			//Surplus
			IF bSurplusAvailable AND Lynus_Standards.GVL_Energy.stDataElectricHeatingElements[diNrOfEMS_OUT,arrCTCheckActivePrio[3]].byPriority = arrActualPrioInTurn[3] AND NOT Lynus_Standards.GVL_Energy.stDataElectricHeatingElements[diNrOfEMS_OUT,arrCTCheckActivePrio[3]].bIsStepSwitched AND NOT 
				Lynus_Standards.GVL_Energy.stDataElectricHeatingElements[diNrOfEMS_OUT,arrCTCheckActivePrio[3]].bIsControllable AND Lynus_Standards.GVL_Energy.stDataElectricHeatingElements[diNrOfEMS_OUT,arrCTCheckActivePrio[3]].arrTargetPowerEMS[1] < 100 THEN
					arrActualStepInTurn[2] := 1;	
						arrMaxPrioReached[3] := FALSE;
							arrMinPrioReached[3] := FALSE;
								arrCTCheckActivePrio[3] := 0;
									uiState := 90;
			ELSIF bSurplusAvailable AND Lynus_Standards.GVL_Energy.stDataElectricHeatingElements[diNrOfEMS_OUT,arrCTCheckActivePrio[3]].byPriority = arrActualPrioInTurn[3] AND Lynus_Standards.GVL_Energy.stDataElectricHeatingElements[diNrOfEMS_OUT,arrCTCheckActivePrio[3]].byNumberOfSteps = 0 AND
				Lynus_Standards.GVL_Energy.stDataElectricHeatingElements[diNrOfEMS_OUT,arrCTCheckActivePrio[3]].arrTargetPowerEMS[1] < 100 THEN 
					arrActualStepInTurn[2] := 1;	
						arrMaxPrioReached[3] := FALSE;
							arrMinPrioReached[3] := FALSE;
								arrCTCheckActivePrio[3] := 0;
									uiState := 90;
			ELSIF bSurplusAvailable AND Lynus_Standards.GVL_Energy.stDataElectricHeatingElements[diNrOfEMS_OUT,arrCTCheckActivePrio[3]].byPriority = arrActualPrioInTurn[3] AND NOT Lynus_Standards.GVL_Energy.stDataElectricHeatingElements[diNrOfEMS_OUT,arrCTCheckActivePrio[3]].bIsStepSwitched AND 
				Lynus_Standards.GVL_Energy.stDataElectricHeatingElements[diNrOfEMS_OUT,arrCTCheckActivePrio[3]].bIsControllable AND Lynus_Standards.GVL_Energy.stDataElectricHeatingElements[diNrOfEMS_OUT,arrCTCheckActivePrio[3]].arrTargetPowerEMS[1] < 100 THEN
					arrActualStepInTurn[2] := 1;	
						arrMaxPrioReached[3] := FALSE;
							arrMinPrioReached[3] := FALSE;
								arrCTCheckActivePrio[3] := 0;
									uiState := 90;	
			ELSIF bSurplusAvailable AND Lynus_Standards.GVL_Energy.stDataElectricHeatingElements[diNrOfEMS_OUT,arrCTCheckActivePrio[3]].byPriority = arrActualPrioInTurn[3] AND Lynus_Standards.GVL_Energy.stDataElectricHeatingElements[diNrOfEMS_OUT,arrCTCheckActivePrio[3]].bIsStepSwitched AND 
				Lynus_Standards.GVL_Energy.stDataElectricHeatingElements[diNrOfEMS_OUT,arrCTCheckActivePrio[3]].bIsControllable AND Lynus_Standards.GVL_Energy.stDataElectricHeatingElements[diNrOfEMS_OUT,arrCTCheckActivePrio[3]].byNumberOfSteps = 1 AND Lynus_Standards.GVL_Energy.stDataElectricHeatingElements[diNrOfEMS_OUT,arrCTCheckActivePrio[3]].arrTargetPowerEMS[1] < 100 THEN 
					arrActualStepInTurn[2] := 1;	
						arrMaxPrioReached[3] := FALSE;
							arrMinPrioReached[3] := FALSE;
								arrCTCheckActivePrio[3] := 0;
									uiState := 90;
			ELSIF bSurplusAvailable AND Lynus_Standards.GVL_Energy.stDataElectricHeatingElements[diNrOfEMS_OUT,arrCTCheckActivePrio[3]].byPriority = arrActualPrioInTurn[3] AND Lynus_Standards.GVL_Energy.stDataElectricHeatingElements[diNrOfEMS_OUT,arrCTCheckActivePrio[3]].bIsStepSwitched AND 
				Lynus_Standards.GVL_Energy.stDataElectricHeatingElements[diNrOfEMS_OUT,arrCTCheckActivePrio[3]].bIsControllable AND Lynus_Standards.GVL_Energy.stDataElectricHeatingElements[diNrOfEMS_OUT,arrCTCheckActivePrio[3]].byNumberOfSteps = 2 AND (Lynus_Standards.GVL_Energy.stDataElectricHeatingElements[diNrOfEMS_OUT,arrCTCheckActivePrio[3]].arrTargetPowerEMS[1] < 100 OR Lynus_Standards.GVL_Energy.stDataElectricHeatingElements[diNrOfEMS_OUT,arrCTCheckActivePrio[3]].arrTargetPowerEMS[2] < 100) THEN
					IF Lynus_Standards.GVL_Energy.stDataElectricHeatingElements[diNrOfEMS_OUT,arrCTCheckActivePrio[3]].arrTargetPowerEMS[1] >= 100 THEN arrActualStepInTurn[2] := 2; ELSE arrActualStepInTurn[2] := 1; END_IF
						arrMaxPrioReached[3] := FALSE;
							arrMinPrioReached[3] := FALSE;
								arrCTCheckActivePrio[3] := 0;
									uiState := 90;
			ELSIF bSurplusAvailable AND Lynus_Standards.GVL_Energy.stDataElectricHeatingElements[diNrOfEMS_OUT,arrCTCheckActivePrio[3]].byPriority = arrActualPrioInTurn[3] AND Lynus_Standards.GVL_Energy.stDataElectricHeatingElements[diNrOfEMS_OUT,arrCTCheckActivePrio[3]].bIsStepSwitched AND 
				Lynus_Standards.GVL_Energy.stDataElectricHeatingElements[diNrOfEMS_OUT,arrCTCheckActivePrio[3]].bIsControllable AND Lynus_Standards.GVL_Energy.stDataElectricHeatingElements[diNrOfEMS_OUT,arrCTCheckActivePrio[3]].byNumberOfSteps = 3 AND (Lynus_Standards.GVL_Energy.stDataElectricHeatingElements[diNrOfEMS_OUT,arrCTCheckActivePrio[3]].arrTargetPowerEMS[1] < 100 OR Lynus_Standards.GVL_Energy.stDataElectricHeatingElements[diNrOfEMS_OUT,arrCTCheckActivePrio[3]].arrTargetPowerEMS[2] < 100 OR Lynus_Standards.GVL_Energy.stDataElectricHeatingElements[diNrOfEMS_OUT,arrCTCheckActivePrio[3]].arrTargetPowerEMS[3] < 100) THEN
					IF Lynus_Standards.GVL_Energy.stDataElectricHeatingElements[diNrOfEMS_OUT,arrCTCheckActivePrio[3]].arrTargetPowerEMS[1] < 100 THEN arrActualStepInTurn[2] := 1; END_IF
					IF Lynus_Standards.GVL_Energy.stDataElectricHeatingElements[diNrOfEMS_OUT,arrCTCheckActivePrio[3]].arrTargetPowerEMS[1] >= 100 THEN arrActualStepInTurn[2] := 2; END_IF
					IF Lynus_Standards.GVL_Energy.stDataElectricHeatingElements[diNrOfEMS_OUT,arrCTCheckActivePrio[3]].arrTargetPowerEMS[2] >= 100 THEN arrActualStepInTurn[2] := 3; END_IF
						arrMaxPrioReached[3] := FALSE;
							arrMinPrioReached[3] := FALSE;
								arrCTCheckActivePrio[3] := 0;
									uiState := 90;
			ELSIF bSurplusAvailable AND Lynus_Standards.GVL_Energy.stDataElectricHeatingElements[diNrOfEMS_OUT,arrCTCheckActivePrio[3]].byPriority = arrActualPrioInTurn[3] AND Lynus_Standards.GVL_Energy.stDataElectricHeatingElements[diNrOfEMS_OUT,arrCTCheckActivePrio[3]].bIsStepSwitched AND 
				Lynus_Standards.GVL_Energy.stDataElectricHeatingElements[diNrOfEMS_OUT,arrCTCheckActivePrio[3]].bIsControllable AND Lynus_Standards.GVL_Energy.stDataElectricHeatingElements[diNrOfEMS_OUT,arrCTCheckActivePrio[3]].byNumberOfSteps = 4 AND 
					(Lynus_Standards.GVL_Energy.stDataElectricHeatingElements[diNrOfEMS_OUT,arrCTCheckActivePrio[3]].arrTargetPowerEMS[1] < 100 OR Lynus_Standards.GVL_Energy.stDataElectricHeatingElements[diNrOfEMS_OUT,arrCTCheckActivePrio[3]].arrTargetPowerEMS[2] < 100 OR Lynus_Standards.GVL_Energy.stDataElectricHeatingElements[diNrOfEMS_OUT,arrCTCheckActivePrio[3]].arrTargetPowerEMS[3] < 100 OR
						Lynus_Standards.GVL_Energy.stDataElectricHeatingElements[diNrOfEMS_OUT,arrCTCheckActivePrio[3]].arrTargetPowerEMS[4] < 100) THEN
							IF Lynus_Standards.GVL_Energy.stDataElectricHeatingElements[diNrOfEMS_OUT,arrCTCheckActivePrio[3]].arrTargetPowerEMS[1] < 100 THEN arrActualStepInTurn[2] := 1; END_IF
							IF Lynus_Standards.GVL_Energy.stDataElectricHeatingElements[diNrOfEMS_OUT,arrCTCheckActivePrio[3]].arrTargetPowerEMS[1] >= 100 THEN arrActualStepInTurn[2] := 2; END_IF
							IF Lynus_Standards.GVL_Energy.stDataElectricHeatingElements[diNrOfEMS_OUT,arrCTCheckActivePrio[3]].arrTargetPowerEMS[2] >= 100 THEN arrActualStepInTurn[2] := 3; END_IF
							IF Lynus_Standards.GVL_Energy.stDataElectricHeatingElements[diNrOfEMS_OUT,arrCTCheckActivePrio[3]].arrTargetPowerEMS[3] >= 100 THEN arrActualStepInTurn[2] := 4; END_IF
								arrMaxPrioReached[3] := FALSE;
									arrMinPrioReached[3] := FALSE;
										arrCTCheckActivePrio[3] := 0;
											uiState := 90;
			ELSIF bSurplusAvailable AND Lynus_Standards.GVL_Energy.stDataElectricHeatingElements[diNrOfEMS_OUT,arrCTCheckActivePrio[3]].byPriority = arrActualPrioInTurn[3] AND Lynus_Standards.GVL_Energy.stDataElectricHeatingElements[diNrOfEMS_OUT,arrCTCheckActivePrio[3]].bIsStepSwitched AND 
				Lynus_Standards.GVL_Energy.stDataElectricHeatingElements[diNrOfEMS_OUT,arrCTCheckActivePrio[3]].bIsControllable AND Lynus_Standards.GVL_Energy.stDataElectricHeatingElements[diNrOfEMS_OUT,arrCTCheckActivePrio[3]].byNumberOfSteps = 5 AND 
					(Lynus_Standards.GVL_Energy.stDataElectricHeatingElements[diNrOfEMS_OUT,arrCTCheckActivePrio[3]].arrTargetPowerEMS[1] < 100 OR Lynus_Standards.GVL_Energy.stDataElectricHeatingElements[diNrOfEMS_OUT,arrCTCheckActivePrio[3]].arrTargetPowerEMS[2] < 100 OR Lynus_Standards.GVL_Energy.stDataElectricHeatingElements[diNrOfEMS_OUT,arrCTCheckActivePrio[3]].arrTargetPowerEMS[3] < 100 OR
						Lynus_Standards.GVL_Energy.stDataElectricHeatingElements[diNrOfEMS_OUT,arrCTCheckActivePrio[3]].arrTargetPowerEMS[4] < 100 OR Lynus_Standards.GVL_Energy.stDataElectricHeatingElements[diNrOfEMS_OUT,arrCTCheckActivePrio[3]].arrTargetPowerEMS[5] < 100) THEN
							IF Lynus_Standards.GVL_Energy.stDataElectricHeatingElements[diNrOfEMS_OUT,arrCTCheckActivePrio[3]].arrTargetPowerEMS[1] < 100 THEN arrActualStepInTurn[2] := 1; END_IF
							IF Lynus_Standards.GVL_Energy.stDataElectricHeatingElements[diNrOfEMS_OUT,arrCTCheckActivePrio[3]].arrTargetPowerEMS[1] >= 100 THEN arrActualStepInTurn[2] := 2; END_IF
							IF Lynus_Standards.GVL_Energy.stDataElectricHeatingElements[diNrOfEMS_OUT,arrCTCheckActivePrio[3]].arrTargetPowerEMS[2] >= 100 THEN arrActualStepInTurn[2] := 3; END_IF
							IF Lynus_Standards.GVL_Energy.stDataElectricHeatingElements[diNrOfEMS_OUT,arrCTCheckActivePrio[3]].arrTargetPowerEMS[3] >= 100 THEN arrActualStepInTurn[2] := 4; END_IF
							IF Lynus_Standards.GVL_Energy.stDataElectricHeatingElements[diNrOfEMS_OUT,arrCTCheckActivePrio[3]].arrTargetPowerEMS[4] >= 100 THEN arrActualStepInTurn[2] := 5; END_IF
								arrMaxPrioReached[3] := FALSE;
									arrMinPrioReached[3] := FALSE;
										arrCTCheckActivePrio[3] := 0;
											uiState := 90;
			ELSIF bSurplusAvailable AND Lynus_Standards.GVL_Energy.stDataElectricHeatingElements[diNrOfEMS_OUT,arrCTCheckActivePrio[3]].byPriority = arrActualPrioInTurn[3] AND Lynus_Standards.GVL_Energy.stDataElectricHeatingElements[diNrOfEMS_OUT,arrCTCheckActivePrio[3]].bIsStepSwitched AND 
				Lynus_Standards.GVL_Energy.stDataElectricHeatingElements[diNrOfEMS_OUT,arrCTCheckActivePrio[3]].bIsControllable AND Lynus_Standards.GVL_Energy.stDataElectricHeatingElements[diNrOfEMS_OUT,arrCTCheckActivePrio[3]].byNumberOfSteps = 6 AND 
					(Lynus_Standards.GVL_Energy.stDataElectricHeatingElements[diNrOfEMS_OUT,arrCTCheckActivePrio[3]].arrTargetPowerEMS[1] < 100 OR Lynus_Standards.GVL_Energy.stDataElectricHeatingElements[diNrOfEMS_OUT,arrCTCheckActivePrio[3]].arrTargetPowerEMS[2]< 100 OR Lynus_Standards.GVL_Energy.stDataElectricHeatingElements[diNrOfEMS_OUT,arrCTCheckActivePrio[3]].arrTargetPowerEMS[3]< 100 OR
						Lynus_Standards.GVL_Energy.stDataElectricHeatingElements[diNrOfEMS_OUT,arrCTCheckActivePrio[3]].arrTargetPowerEMS[4] < 100 OR Lynus_Standards.GVL_Energy.stDataElectricHeatingElements[diNrOfEMS_OUT,arrCTCheckActivePrio[3]].arrTargetPowerEMS[5] < 100 OR Lynus_Standards.GVL_Energy.stDataElectricHeatingElements[diNrOfEMS_OUT,arrCTCheckActivePrio[3]].arrTargetPowerEMS[6] < 100) THEN
							IF Lynus_Standards.GVL_Energy.stDataElectricHeatingElements[diNrOfEMS_OUT,arrCTCheckActivePrio[3]].arrTargetPowerEMS[1] < 100 THEN arrActualStepInTurn[2] := 1; END_IF
							IF Lynus_Standards.GVL_Energy.stDataElectricHeatingElements[diNrOfEMS_OUT,arrCTCheckActivePrio[3]].arrTargetPowerEMS[1] >= 100 THEN arrActualStepInTurn[2] := 2; END_IF
							IF Lynus_Standards.GVL_Energy.stDataElectricHeatingElements[diNrOfEMS_OUT,arrCTCheckActivePrio[3]].arrTargetPowerEMS[2] >= 100 THEN arrActualStepInTurn[2] := 3; END_IF
							IF Lynus_Standards.GVL_Energy.stDataElectricHeatingElements[diNrOfEMS_OUT,arrCTCheckActivePrio[3]].arrTargetPowerEMS[3] >= 100 THEN arrActualStepInTurn[2] := 4; END_IF
							IF Lynus_Standards.GVL_Energy.stDataElectricHeatingElements[diNrOfEMS_OUT,arrCTCheckActivePrio[3]].arrTargetPowerEMS[4] >= 100 THEN arrActualStepInTurn[2] := 5; END_IF
							IF Lynus_Standards.GVL_Energy.stDataElectricHeatingElements[diNrOfEMS_OUT,arrCTCheckActivePrio[3]].arrTargetPowerEMS[5] >= 100 THEN arrActualStepInTurn[2] := 6; END_IF
								arrMaxPrioReached[3] := FALSE;
									arrMinPrioReached[3] := FALSE;
										arrCTCheckActivePrio[3] := 0;
											uiState := 90;
			ELSIF bSurplusAvailable AND Lynus_Standards.GVL_Energy.stDataElectricHeatingElements[diNrOfEMS_OUT,arrCTCheckActivePrio[3]].byPriority = arrActualPrioInTurn[3] AND Lynus_Standards.GVL_Energy.stDataElectricHeatingElements[diNrOfEMS_OUT,arrCTCheckActivePrio[3]].bIsStepSwitched AND 
				Lynus_Standards.GVL_Energy.stDataElectricHeatingElements[diNrOfEMS_OUT,arrCTCheckActivePrio[3]].bIsControllable AND Lynus_Standards.GVL_Energy.stDataElectricHeatingElements[diNrOfEMS_OUT,arrCTCheckActivePrio[3]].byNumberOfSteps= 7 AND 
					(Lynus_Standards.GVL_Energy.stDataElectricHeatingElements[diNrOfEMS_OUT,arrCTCheckActivePrio[3]].arrTargetPowerEMS[1] < 100 OR Lynus_Standards.GVL_Energy.stDataElectricHeatingElements[diNrOfEMS_OUT,arrCTCheckActivePrio[3]].arrTargetPowerEMS[2] < 100 OR Lynus_Standards.GVL_Energy.stDataElectricHeatingElements[diNrOfEMS_OUT,arrCTCheckActivePrio[3]].arrTargetPowerEMS[3] < 100 OR
						Lynus_Standards.GVL_Energy.stDataElectricHeatingElements[diNrOfEMS_OUT,arrCTCheckActivePrio[3]].arrTargetPowerEMS[4] < 100 OR Lynus_Standards.GVL_Energy.stDataElectricHeatingElements[diNrOfEMS_OUT,arrCTCheckActivePrio[3]].arrTargetPowerEMS[5] < 100 OR Lynus_Standards.GVL_Energy.stDataElectricHeatingElements[diNrOfEMS_OUT,arrCTCheckActivePrio[3]].arrTargetPowerEMS[6] < 100 OR
							Lynus_Standards.GVL_Energy.stDataElectricHeatingElements[diNrOfEMS_OUT,arrCTCheckActivePrio[3]].arrTargetPowerEMS[7] < 100) THEN
								IF Lynus_Standards.GVL_Energy.stDataElectricHeatingElements[diNrOfEMS_OUT,arrCTCheckActivePrio[3]].arrTargetPowerEMS[1] < 100 THEN arrActualStepInTurn[2] := 1; END_IF
								IF Lynus_Standards.GVL_Energy.stDataElectricHeatingElements[diNrOfEMS_OUT,arrCTCheckActivePrio[3]].arrTargetPowerEMS[1] >= 100 THEN arrActualStepInTurn[2] := 2; END_IF
								IF Lynus_Standards.GVL_Energy.stDataElectricHeatingElements[diNrOfEMS_OUT,arrCTCheckActivePrio[3]].arrTargetPowerEMS[2] >= 100 THEN arrActualStepInTurn[2] := 3; END_IF
								IF Lynus_Standards.GVL_Energy.stDataElectricHeatingElements[diNrOfEMS_OUT,arrCTCheckActivePrio[3]].arrTargetPowerEMS[3] >= 100 THEN arrActualStepInTurn[2] := 4; END_IF
								IF Lynus_Standards.GVL_Energy.stDataElectricHeatingElements[diNrOfEMS_OUT,arrCTCheckActivePrio[3]].arrTargetPowerEMS[4] >= 100 THEN arrActualStepInTurn[2] := 5; END_IF
								IF Lynus_Standards.GVL_Energy.stDataElectricHeatingElements[diNrOfEMS_OUT,arrCTCheckActivePrio[3]].arrTargetPowerEMS[5] >= 100 THEN arrActualStepInTurn[2] := 6; END_IF
								IF Lynus_Standards.GVL_Energy.stDataElectricHeatingElements[diNrOfEMS_OUT,arrCTCheckActivePrio[3]].arrTargetPowerEMS[6] >= 100 THEN arrActualStepInTurn[2] := 7; END_IF
									arrMaxPrioReached[3] := FALSE;
										arrMinPrioReached[3] := FALSE;
											arrCTCheckActivePrio[3] := 0;
												uiState := 90;
			ELSIF bSurplusAvailable AND Lynus_Standards.GVL_Energy.stDataElectricHeatingElements[diNrOfEMS_OUT,arrCTCheckActivePrio[3]].byPriority = arrActualPrioInTurn[3] AND Lynus_Standards.GVL_Energy.stDataElectricHeatingElements[diNrOfEMS_OUT,arrCTCheckActivePrio[3]].bIsStepSwitched AND 
				Lynus_Standards.GVL_Energy.stDataElectricHeatingElements[diNrOfEMS_OUT,arrCTCheckActivePrio[3]].bIsControllable AND Lynus_Standards.GVL_Energy.stDataElectricHeatingElements[diNrOfEMS_OUT,arrCTCheckActivePrio[3]].byNumberOfSteps = 8 AND 
					(Lynus_Standards.GVL_Energy.stDataElectricHeatingElements[diNrOfEMS_OUT,arrCTCheckActivePrio[3]].arrTargetPowerEMS[1] < 100 OR Lynus_Standards.GVL_Energy.stDataElectricHeatingElements[diNrOfEMS_OUT,arrCTCheckActivePrio[3]].arrTargetPowerEMS[2] < 100 OR Lynus_Standards.GVL_Energy.stDataElectricHeatingElements[diNrOfEMS_OUT,arrCTCheckActivePrio[3]].arrTargetPowerEMS[3] < 100 OR
						Lynus_Standards.GVL_Energy.stDataElectricHeatingElements[diNrOfEMS_OUT,arrCTCheckActivePrio[3]].arrTargetPowerEMS[4] < 100 OR Lynus_Standards.GVL_Energy.stDataElectricHeatingElements[diNrOfEMS_OUT,arrCTCheckActivePrio[3]].arrTargetPowerEMS[5] < 100 OR Lynus_Standards.GVL_Energy.stDataElectricHeatingElements[diNrOfEMS_OUT,arrCTCheckActivePrio[3]].arrTargetPowerEMS[6] < 100 OR
							Lynus_Standards.GVL_Energy.stDataElectricHeatingElements[diNrOfEMS_OUT,arrCTCheckActivePrio[3]].arrTargetPowerEMS[7] < 100 OR Lynus_Standards.GVL_Energy.stDataElectricHeatingElements[diNrOfEMS_OUT,arrCTCheckActivePrio[3]].arrTargetPowerEMS[8] < 100) THEN
								IF Lynus_Standards.GVL_Energy.stDataElectricHeatingElements[diNrOfEMS_OUT,arrCTCheckActivePrio[3]].arrTargetPowerEMS[1] < 100 THEN arrActualStepInTurn[2] := 1; END_IF
								IF Lynus_Standards.GVL_Energy.stDataElectricHeatingElements[diNrOfEMS_OUT,arrCTCheckActivePrio[3]].arrTargetPowerEMS[1] >= 100 THEN arrActualStepInTurn[2] := 2; END_IF
								IF Lynus_Standards.GVL_Energy.stDataElectricHeatingElements[diNrOfEMS_OUT,arrCTCheckActivePrio[3]].arrTargetPowerEMS[2] >= 100 THEN arrActualStepInTurn[2] := 3; END_IF
								IF Lynus_Standards.GVL_Energy.stDataElectricHeatingElements[diNrOfEMS_OUT,arrCTCheckActivePrio[3]].arrTargetPowerEMS[3] >= 100 THEN arrActualStepInTurn[2] := 4; END_IF
								IF Lynus_Standards.GVL_Energy.stDataElectricHeatingElements[diNrOfEMS_OUT,arrCTCheckActivePrio[3]].arrTargetPowerEMS[4] >= 100 THEN arrActualStepInTurn[2] := 5; END_IF
								IF Lynus_Standards.GVL_Energy.stDataElectricHeatingElements[diNrOfEMS_OUT,arrCTCheckActivePrio[3]].arrTargetPowerEMS[5] >= 100 THEN arrActualStepInTurn[2] := 6; END_IF
								IF Lynus_Standards.GVL_Energy.stDataElectricHeatingElements[diNrOfEMS_OUT,arrCTCheckActivePrio[3]].arrTargetPowerEMS[6] >= 100 THEN arrActualStepInTurn[2] := 7; END_IF
								IF Lynus_Standards.GVL_Energy.stDataElectricHeatingElements[diNrOfEMS_OUT,arrCTCheckActivePrio[3]].arrTargetPowerEMS[7] >= 100 THEN arrActualStepInTurn[2] := 8; END_IF
									arrMaxPrioReached[3] := FALSE;
										arrMinPrioReached[3] := FALSE;
											arrCTCheckActivePrio[3] := 0;
												uiState := 90;
			ELSIF bSurplusAvailable AND Lynus_Standards.GVL_Energy.stDataElectricHeatingElements[diNrOfEMS_OUT,arrCTCheckActivePrio[3]].byPriority = arrActualPrioInTurn[3] AND Lynus_Standards.GVL_Energy.stDataElectricHeatingElements[diNrOfEMS_OUT,arrCTCheckActivePrio[3]].bIsStepSwitched AND 
				Lynus_Standards.GVL_Energy.stDataElectricHeatingElements[diNrOfEMS_OUT,arrCTCheckActivePrio[3]].bIsControllable AND Lynus_Standards.GVL_Energy.stDataElectricHeatingElements[diNrOfEMS_OUT,arrCTCheckActivePrio[3]].byNumberOfSteps = 9 AND 
					(Lynus_Standards.GVL_Energy.stDataElectricHeatingElements[diNrOfEMS_OUT,arrCTCheckActivePrio[3]].arrTargetPowerEMS[1] < 100 OR Lynus_Standards.GVL_Energy.stDataElectricHeatingElements[diNrOfEMS_OUT,arrCTCheckActivePrio[3]].arrTargetPowerEMS[2] < 100 OR Lynus_Standards.GVL_Energy.stDataElectricHeatingElements[diNrOfEMS_OUT,arrCTCheckActivePrio[3]].arrTargetPowerEMS[3] < 100 OR
						Lynus_Standards.GVL_Energy.stDataElectricHeatingElements[diNrOfEMS_OUT,arrCTCheckActivePrio[3]].arrTargetPowerEMS[4] < 100 OR Lynus_Standards.GVL_Energy.stDataElectricHeatingElements[diNrOfEMS_OUT,arrCTCheckActivePrio[3]].arrTargetPowerEMS[5] < 100 OR Lynus_Standards.GVL_Energy.stDataElectricHeatingElements[diNrOfEMS_OUT,arrCTCheckActivePrio[3]].arrTargetPowerEMS[6] < 100 OR
							Lynus_Standards.GVL_Energy.stDataElectricHeatingElements[diNrOfEMS_OUT,arrCTCheckActivePrio[3]].arrTargetPowerEMS[7] < 100 OR Lynus_Standards.GVL_Energy.stDataElectricHeatingElements[diNrOfEMS_OUT,arrCTCheckActivePrio[3]].arrTargetPowerEMS[8] < 100 OR Lynus_Standards.GVL_Energy.stDataElectricHeatingElements[diNrOfEMS_OUT,arrCTCheckActivePrio[3]].arrTargetPowerEMS[9] < 100) THEN
								IF Lynus_Standards.GVL_Energy.stDataElectricHeatingElements[diNrOfEMS_OUT,arrCTCheckActivePrio[3]].arrTargetPowerEMS[1] < 100 THEN arrActualStepInTurn[2] := 1; END_IF
								IF Lynus_Standards.GVL_Energy.stDataElectricHeatingElements[diNrOfEMS_OUT,arrCTCheckActivePrio[3]].arrTargetPowerEMS[1] >= 100 THEN arrActualStepInTurn[2] := 2; END_IF
								IF Lynus_Standards.GVL_Energy.stDataElectricHeatingElements[diNrOfEMS_OUT,arrCTCheckActivePrio[3]].arrTargetPowerEMS[2] >= 100 THEN arrActualStepInTurn[2] := 3; END_IF
								IF Lynus_Standards.GVL_Energy.stDataElectricHeatingElements[diNrOfEMS_OUT,arrCTCheckActivePrio[3]].arrTargetPowerEMS[3] >= 100 THEN arrActualStepInTurn[2] := 4; END_IF
								IF Lynus_Standards.GVL_Energy.stDataElectricHeatingElements[diNrOfEMS_OUT,arrCTCheckActivePrio[3]].arrTargetPowerEMS[4] >= 100 THEN arrActualStepInTurn[2] := 5; END_IF
								IF Lynus_Standards.GVL_Energy.stDataElectricHeatingElements[diNrOfEMS_OUT,arrCTCheckActivePrio[3]].arrTargetPowerEMS[5] >= 100 THEN arrActualStepInTurn[2] := 6; END_IF
								IF Lynus_Standards.GVL_Energy.stDataElectricHeatingElements[diNrOfEMS_OUT,arrCTCheckActivePrio[3]].arrTargetPowerEMS[6] >= 100 THEN arrActualStepInTurn[2] := 7; END_IF
								IF Lynus_Standards.GVL_Energy.stDataElectricHeatingElements[diNrOfEMS_OUT,arrCTCheckActivePrio[3]].arrTargetPowerEMS[7] >= 100 THEN arrActualStepInTurn[2] := 8; END_IF
								IF Lynus_Standards.GVL_Energy.stDataElectricHeatingElements[diNrOfEMS_OUT,arrCTCheckActivePrio[3]].arrTargetPowerEMS[8] >= 100 THEN arrActualStepInTurn[2] := 9; END_IF
									arrMaxPrioReached[3] := FALSE;
										arrMinPrioReached[3] := FALSE;
											arrCTCheckActivePrio[3] := 0;
												uiState := 90;
			ELSIF bSurplusAvailable AND Lynus_Standards.GVL_Energy.stDataElectricHeatingElements[diNrOfEMS_OUT,arrCTCheckActivePrio[3]].byPriority = arrActualPrioInTurn[3] AND Lynus_Standards.GVL_Energy.stDataElectricHeatingElements[diNrOfEMS_OUT,arrCTCheckActivePrio[3]].bIsStepSwitched AND 
				Lynus_Standards.GVL_Energy.stDataElectricHeatingElements[diNrOfEMS_OUT,arrCTCheckActivePrio[3]].bIsControllable AND Lynus_Standards.GVL_Energy.stDataElectricHeatingElements[diNrOfEMS_OUT,arrCTCheckActivePrio[3]].byNumberOfSteps = 10 AND 
					(Lynus_Standards.GVL_Energy.stDataElectricHeatingElements[diNrOfEMS_OUT,arrCTCheckActivePrio[3]].arrTargetPowerEMS[1] < 100 OR Lynus_Standards.GVL_Energy.stDataElectricHeatingElements[diNrOfEMS_OUT,arrCTCheckActivePrio[3]].arrTargetPowerEMS[2] < 100 OR Lynus_Standards.GVL_Energy.stDataElectricHeatingElements[diNrOfEMS_OUT,arrCTCheckActivePrio[3]].arrTargetPowerEMS[3] < 100 OR
						Lynus_Standards.GVL_Energy.stDataElectricHeatingElements[diNrOfEMS_OUT,arrCTCheckActivePrio[3]].arrTargetPowerEMS[4] < 100 OR Lynus_Standards.GVL_Energy.stDataElectricHeatingElements[diNrOfEMS_OUT,arrCTCheckActivePrio[3]].arrTargetPowerEMS[5] < 100 OR Lynus_Standards.GVL_Energy.stDataElectricHeatingElements[diNrOfEMS_OUT,arrCTCheckActivePrio[3]].arrTargetPowerEMS[6] < 100 OR
							Lynus_Standards.GVL_Energy.stDataElectricHeatingElements[diNrOfEMS_OUT,arrCTCheckActivePrio[3]].arrTargetPowerEMS[7] < 100 OR Lynus_Standards.GVL_Energy.stDataElectricHeatingElements[diNrOfEMS_OUT,arrCTCheckActivePrio[3]].arrTargetPowerEMS[8] < 100 OR Lynus_Standards.GVL_Energy.stDataElectricHeatingElements[diNrOfEMS_OUT,arrCTCheckActivePrio[3]].arrTargetPowerEMS[9] < 100 OR
								Lynus_Standards.GVL_Energy.stDataElectricHeatingElements[diNrOfEMS_OUT,arrCTCheckActivePrio[3]].arrTargetPowerEMS[10] < 100) THEN
									IF Lynus_Standards.GVL_Energy.stDataElectricHeatingElements[diNrOfEMS_OUT,arrCTCheckActivePrio[3]].arrTargetPowerEMS[1] < 100 THEN arrActualStepInTurn[2] := 1; END_IF
									IF Lynus_Standards.GVL_Energy.stDataElectricHeatingElements[diNrOfEMS_OUT,arrCTCheckActivePrio[3]].arrTargetPowerEMS[1] >= 100 THEN arrActualStepInTurn[2] := 2; END_IF
									IF Lynus_Standards.GVL_Energy.stDataElectricHeatingElements[diNrOfEMS_OUT,arrCTCheckActivePrio[3]].arrTargetPowerEMS[2] >= 100 THEN arrActualStepInTurn[2] := 3; END_IF
									IF Lynus_Standards.GVL_Energy.stDataElectricHeatingElements[diNrOfEMS_OUT,arrCTCheckActivePrio[3]].arrTargetPowerEMS[3] >= 100 THEN arrActualStepInTurn[2] := 4; END_IF
									IF Lynus_Standards.GVL_Energy.stDataElectricHeatingElements[diNrOfEMS_OUT,arrCTCheckActivePrio[3]].arrTargetPowerEMS[4] >= 100 THEN arrActualStepInTurn[2] := 5; END_IF
									IF Lynus_Standards.GVL_Energy.stDataElectricHeatingElements[diNrOfEMS_OUT,arrCTCheckActivePrio[3]].arrTargetPowerEMS[5] >= 100 THEN arrActualStepInTurn[2] := 6; END_IF
									IF Lynus_Standards.GVL_Energy.stDataElectricHeatingElements[diNrOfEMS_OUT,arrCTCheckActivePrio[3]].arrTargetPowerEMS[6] >= 100 THEN arrActualStepInTurn[2] := 7; END_IF
									IF Lynus_Standards.GVL_Energy.stDataElectricHeatingElements[diNrOfEMS_OUT,arrCTCheckActivePrio[3]].arrTargetPowerEMS[7] >= 100 THEN arrActualStepInTurn[2] := 8; END_IF
									IF Lynus_Standards.GVL_Energy.stDataElectricHeatingElements[diNrOfEMS_OUT,arrCTCheckActivePrio[3]].arrTargetPowerEMS[8] >= 100 THEN arrActualStepInTurn[2] := 9; END_IF
									IF Lynus_Standards.GVL_Energy.stDataElectricHeatingElements[diNrOfEMS_OUT,arrCTCheckActivePrio[3]].arrTargetPowerEMS[9] >= 100 THEN arrActualStepInTurn[2] := 10; END_IF
										arrMaxPrioReached[3] := FALSE;
											arrMinPrioReached[3] := FALSE;
												arrCTCheckActivePrio[3] := 0;
													uiState := 90;
			ELSE
				IF bSurplusAvailable AND arrActualPrioInTurn[3] < 255 AND uiState = 70 AND arrCTCheckActivePrio[3] = Constants_Energy.diMaxNumberOfElectricHeatingElements THEN 
					arrActualPrioInTurn[3] := arrActualPrioInTurn[3] + 1; arrCTCheckActivePrio[3] := 0; liCounterCkeckDeviceAndPrio := 0; liNrOfNotDoneDevices := 0; 
				END_IF
			END_IF
				//No surplus
				IF NOT bSurplusAvailable AND Lynus_Standards.GVL_Energy.stDataElectricHeatingElements[diNrOfEMS_OUT,arrCTCheckActivePrio[3]].byPriority = arrActualPrioInTurn[3] AND NOT Lynus_Standards.GVL_Energy.stDataElectricHeatingElements[diNrOfEMS_OUT,arrCTCheckActivePrio[3]].bIsStepSwitched AND NOT 
					Lynus_Standards.GVL_Energy.stDataElectricHeatingElements[diNrOfEMS_OUT,arrCTCheckActivePrio[3]].bIsControllable AND Lynus_Standards.GVL_Energy.stDataElectricHeatingElements[diNrOfEMS_OUT,arrCTCheckActivePrio[3]].arrTargetPowerEMS[1] > 0 THEN
						arrActualStepInTurn[2] := 1;	
							arrMaxPrioReached[3] := FALSE;
								arrMinPrioReached[3] := FALSE;
									arrCTCheckActivePrio[3] := 0;
										uiState := 90;
				ELSIF NOT bSurplusAvailable AND Lynus_Standards.GVL_Energy.stDataElectricHeatingElements[diNrOfEMS_OUT,arrCTCheckActivePrio[3]].byPriority = arrActualPrioInTurn[3] AND Lynus_Standards.GVL_Energy.stDataElectricHeatingElements[diNrOfEMS_OUT,arrCTCheckActivePrio[3]].byNumberOfSteps = 0 AND
					Lynus_Standards.GVL_Energy.stDataElectricHeatingElements[diNrOfEMS_OUT,arrCTCheckActivePrio[3]].arrTargetPowerEMS[1] > 0 THEN 
						arrActualStepInTurn[2] := 1;	
							arrMaxPrioReached[3] := FALSE;
								arrMinPrioReached[3] := FALSE;
									arrCTCheckActivePrio[3] := 0;
										uiState := 90;
				ELSIF NOT bSurplusAvailable AND Lynus_Standards.GVL_Energy.stDataElectricHeatingElements[diNrOfEMS_OUT,arrCTCheckActivePrio[3]].byPriority = arrActualPrioInTurn[3] AND NOT Lynus_Standards.GVL_Energy.stDataElectricHeatingElements[diNrOfEMS_OUT,arrCTCheckActivePrio[3]].bIsStepSwitched AND 
					Lynus_Standards.GVL_Energy.stDataElectricHeatingElements[diNrOfEMS_OUT,arrCTCheckActivePrio[3]].bIsControllable AND Lynus_Standards.GVL_Energy.stDataElectricHeatingElements[diNrOfEMS_OUT,arrCTCheckActivePrio[3]].arrTargetPowerEMS[1] > 0 THEN
						arrActualStepInTurn[2] := 1;	
							arrMaxPrioReached[3] := FALSE;
								arrMinPrioReached[3] := FALSE;
									arrCTCheckActivePrio[3] := 0;
										uiState := 90;	
				ELSIF NOT bSurplusAvailable AND Lynus_Standards.GVL_Energy.stDataElectricHeatingElements[diNrOfEMS_OUT,arrCTCheckActivePrio[3]].byPriority = arrActualPrioInTurn[3] AND Lynus_Standards.GVL_Energy.stDataElectricHeatingElements[diNrOfEMS_OUT,arrCTCheckActivePrio[3]].bIsStepSwitched AND 
					Lynus_Standards.GVL_Energy.stDataElectricHeatingElements[diNrOfEMS_OUT,arrCTCheckActivePrio[3]].bIsControllable AND Lynus_Standards.GVL_Energy.stDataElectricHeatingElements[diNrOfEMS_OUT,arrCTCheckActivePrio[3]].byNumberOfSteps = 1 AND Lynus_Standards.GVL_Energy.stDataElectricHeatingElements[diNrOfEMS_OUT,arrCTCheckActivePrio[3]].arrTargetPowerEMS[1] > 0 THEN 
						arrActualStepInTurn[2] := 1;	
							arrMaxPrioReached[3] := FALSE;
								arrMinPrioReached[3] := FALSE;
									arrCTCheckActivePrio[3] := 0;
										uiState := 90;
				ELSIF NOT bSurplusAvailable AND Lynus_Standards.GVL_Energy.stDataElectricHeatingElements[diNrOfEMS_OUT,arrCTCheckActivePrio[3]].byPriority = arrActualPrioInTurn[3] AND Lynus_Standards.GVL_Energy.stDataElectricHeatingElements[diNrOfEMS_OUT,arrCTCheckActivePrio[3]].bIsStepSwitched AND 
					Lynus_Standards.GVL_Energy.stDataElectricHeatingElements[diNrOfEMS_OUT,arrCTCheckActivePrio[3]].bIsControllable AND Lynus_Standards.GVL_Energy.stDataElectricHeatingElements[diNrOfEMS_OUT,arrCTCheckActivePrio[3]].byNumberOfSteps = 2 AND (Lynus_Standards.GVL_Energy.stDataElectricHeatingElements[diNrOfEMS_OUT,arrCTCheckActivePrio[3]].arrTargetPowerEMS[1] > 0 OR Lynus_Standards.GVL_Energy.stDataElectricHeatingElements[diNrOfEMS_OUT,arrCTCheckActivePrio[3]].arrTargetPowerEMS[2] > 0) THEN
						IF Lynus_Standards.GVL_Energy.stDataElectricHeatingElements[diNrOfEMS_OUT,arrCTCheckActivePrio[3]].arrTargetPowerEMS[2] <= 0 THEN arrActualStepInTurn[2] := 1; ELSE arrActualStepInTurn[2] := 2; END_IF
							arrMaxPrioReached[3] := FALSE;
								arrMinPrioReached[3] := FALSE;
									arrCTCheckActivePrio[3] := 0;
										uiState := 90;
				ELSIF NOT bSurplusAvailable AND Lynus_Standards.GVL_Energy.stDataElectricHeatingElements[diNrOfEMS_OUT,arrCTCheckActivePrio[3]].byPriority = arrActualPrioInTurn[3] AND Lynus_Standards.GVL_Energy.stDataElectricHeatingElements[diNrOfEMS_OUT,arrCTCheckActivePrio[3]].bIsStepSwitched AND 
					Lynus_Standards.GVL_Energy.stDataElectricHeatingElements[diNrOfEMS_OUT,arrCTCheckActivePrio[3]].bIsControllable AND Lynus_Standards.GVL_Energy.stDataElectricHeatingElements[diNrOfEMS_OUT,arrCTCheckActivePrio[3]].byNumberOfSteps = 3 AND (Lynus_Standards.GVL_Energy.stDataElectricHeatingElements[diNrOfEMS_OUT,arrCTCheckActivePrio[3]].arrTargetPowerEMS[1] > 0 OR Lynus_Standards.GVL_Energy.stDataElectricHeatingElements[diNrOfEMS_OUT,arrCTCheckActivePrio[3]].arrTargetPowerEMS[2] > 0 OR Lynus_Standards.GVL_Energy.stDataElectricHeatingElements[diNrOfEMS_OUT,arrCTCheckActivePrio[3]].arrTargetPowerEMS[3] > 0) THEN
						IF Lynus_Standards.GVL_Energy.stDataElectricHeatingElements[diNrOfEMS_OUT,arrCTCheckActivePrio[3]].arrTargetPowerEMS[2] <= 0 THEN arrActualStepInTurn[2] := 1; END_IF
						IF Lynus_Standards.GVL_Energy.stDataElectricHeatingElements[diNrOfEMS_OUT,arrCTCheckActivePrio[3]].arrTargetPowerEMS[2] > 0 THEN arrActualStepInTurn[2] := 2; END_IF
						IF Lynus_Standards.GVL_Energy.stDataElectricHeatingElements[diNrOfEMS_OUT,arrCTCheckActivePrio[3]].arrTargetPowerEMS[3] > 0 THEN arrActualStepInTurn[2] := 3; END_IF
							arrMaxPrioReached[3] := FALSE;
								arrMinPrioReached[3] := FALSE;
									arrCTCheckActivePrio[3] := 0;
										uiState := 90;
				ELSIF NOT bSurplusAvailable AND Lynus_Standards.GVL_Energy.stDataElectricHeatingElements[diNrOfEMS_OUT,arrCTCheckActivePrio[3]].byPriority = arrActualPrioInTurn[3] AND Lynus_Standards.GVL_Energy.stDataElectricHeatingElements[diNrOfEMS_OUT,arrCTCheckActivePrio[3]].bIsStepSwitched AND 
					Lynus_Standards.GVL_Energy.stDataElectricHeatingElements[diNrOfEMS_OUT,arrCTCheckActivePrio[3]].bIsControllable AND Lynus_Standards.GVL_Energy.stDataElectricHeatingElements[diNrOfEMS_OUT,arrCTCheckActivePrio[3]].byNumberOfSteps = 4 AND 
						(Lynus_Standards.GVL_Energy.stDataElectricHeatingElements[diNrOfEMS_OUT,arrCTCheckActivePrio[3]].arrTargetPowerEMS[1] > 0 OR Lynus_Standards.GVL_Energy.stDataElectricHeatingElements[diNrOfEMS_OUT,arrCTCheckActivePrio[3]].arrTargetPowerEMS[2] > 0 OR Lynus_Standards.GVL_Energy.stDataElectricHeatingElements[diNrOfEMS_OUT,arrCTCheckActivePrio[3]].arrTargetPowerEMS[3] > 0 OR
							Lynus_Standards.GVL_Energy.stDataElectricHeatingElements[diNrOfEMS_OUT,arrCTCheckActivePrio[3]].arrTargetPowerEMS[4] > 0) THEN
								IF Lynus_Standards.GVL_Energy.stDataElectricHeatingElements[diNrOfEMS_OUT,arrCTCheckActivePrio[3]].arrTargetPowerEMS[2] <= 0 THEN arrActualStepInTurn[2] := 1; END_IF
								IF Lynus_Standards.GVL_Energy.stDataElectricHeatingElements[diNrOfEMS_OUT,arrCTCheckActivePrio[3]].arrTargetPowerEMS[2] > 0 THEN arrActualStepInTurn[2] := 2; END_IF
								IF Lynus_Standards.GVL_Energy.stDataElectricHeatingElements[diNrOfEMS_OUT,arrCTCheckActivePrio[3]].arrTargetPowerEMS[3] > 0 THEN arrActualStepInTurn[2] := 3; END_IF
								IF Lynus_Standards.GVL_Energy.stDataElectricHeatingElements[diNrOfEMS_OUT,arrCTCheckActivePrio[3]].arrTargetPowerEMS[4] > 0 THEN arrActualStepInTurn[2] := 4; END_IF
									arrMaxPrioReached[3] := FALSE;
										arrMinPrioReached[3] := FALSE;
											arrCTCheckActivePrio[3] := 0;
												uiState := 90;
				ELSIF NOT bSurplusAvailable AND Lynus_Standards.GVL_Energy.stDataElectricHeatingElements[diNrOfEMS_OUT,arrCTCheckActivePrio[3]].byPriority = arrActualPrioInTurn[3] AND Lynus_Standards.GVL_Energy.stDataElectricHeatingElements[diNrOfEMS_OUT,arrCTCheckActivePrio[3]].bIsStepSwitched AND 
					Lynus_Standards.GVL_Energy.stDataElectricHeatingElements[diNrOfEMS_OUT,arrCTCheckActivePrio[3]].bIsControllable AND Lynus_Standards.GVL_Energy.stDataElectricHeatingElements[diNrOfEMS_OUT,arrCTCheckActivePrio[3]].byNumberOfSteps = 5 AND 
						(Lynus_Standards.GVL_Energy.stDataElectricHeatingElements[diNrOfEMS_OUT,arrCTCheckActivePrio[3]].arrTargetPowerEMS[1] > 0 OR Lynus_Standards.GVL_Energy.stDataElectricHeatingElements[diNrOfEMS_OUT,arrCTCheckActivePrio[3]].arrTargetPowerEMS[2] > 0 OR Lynus_Standards.GVL_Energy.stDataElectricHeatingElements[diNrOfEMS_OUT,arrCTCheckActivePrio[3]].arrTargetPowerEMS[3] > 0 OR
							Lynus_Standards.GVL_Energy.stDataElectricHeatingElements[diNrOfEMS_OUT,arrCTCheckActivePrio[3]].arrTargetPowerEMS[4] > 0 OR Lynus_Standards.GVL_Energy.stDataElectricHeatingElements[diNrOfEMS_OUT,arrCTCheckActivePrio[3]].arrTargetPowerEMS[5] > 0) THEN
								IF Lynus_Standards.GVL_Energy.stDataElectricHeatingElements[diNrOfEMS_OUT,arrCTCheckActivePrio[3]].arrTargetPowerEMS[2] <= 0 THEN arrActualStepInTurn[2] := 1; END_IF
								IF Lynus_Standards.GVL_Energy.stDataElectricHeatingElements[diNrOfEMS_OUT,arrCTCheckActivePrio[3]].arrTargetPowerEMS[2] > 0 THEN arrActualStepInTurn[2] := 2; END_IF
								IF Lynus_Standards.GVL_Energy.stDataElectricHeatingElements[diNrOfEMS_OUT,arrCTCheckActivePrio[3]].arrTargetPowerEMS[3] > 0 THEN arrActualStepInTurn[2] := 3; END_IF
								IF Lynus_Standards.GVL_Energy.stDataElectricHeatingElements[diNrOfEMS_OUT,arrCTCheckActivePrio[3]].arrTargetPowerEMS[4] > 0 THEN arrActualStepInTurn[2] := 4; END_IF
								IF Lynus_Standards.GVL_Energy.stDataElectricHeatingElements[diNrOfEMS_OUT,arrCTCheckActivePrio[3]].arrTargetPowerEMS[5] > 0 THEN arrActualStepInTurn[2] := 5; END_IF
									arrMaxPrioReached[3] := FALSE;
										arrMinPrioReached[3] := FALSE;
											arrCTCheckActivePrio[3] := 0;
												uiState := 90;
				ELSIF NOT bSurplusAvailable AND Lynus_Standards.GVL_Energy.stDataElectricHeatingElements[diNrOfEMS_OUT,arrCTCheckActivePrio[3]].byPriority = arrActualPrioInTurn[3] AND Lynus_Standards.GVL_Energy.stDataElectricHeatingElements[diNrOfEMS_OUT,arrCTCheckActivePrio[3]].bIsStepSwitched AND 
					Lynus_Standards.GVL_Energy.stDataElectricHeatingElements[diNrOfEMS_OUT,arrCTCheckActivePrio[3]].bIsControllable AND Lynus_Standards.GVL_Energy.stDataElectricHeatingElements[diNrOfEMS_OUT,arrCTCheckActivePrio[3]].byNumberOfSteps = 6 AND 
						(Lynus_Standards.GVL_Energy.stDataElectricHeatingElements[diNrOfEMS_OUT,arrCTCheckActivePrio[3]].arrTargetPowerEMS[1] > 0 OR Lynus_Standards.GVL_Energy.stDataElectricHeatingElements[diNrOfEMS_OUT,arrCTCheckActivePrio[3]].arrTargetPowerEMS[2] > 0 OR Lynus_Standards.GVL_Energy.stDataElectricHeatingElements[diNrOfEMS_OUT,arrCTCheckActivePrio[3]].arrTargetPowerEMS[3] > 0 OR
							Lynus_Standards.GVL_Energy.stDataElectricHeatingElements[diNrOfEMS_OUT,arrCTCheckActivePrio[3]].arrTargetPowerEMS[4] > 0 OR Lynus_Standards.GVL_Energy.stDataElectricHeatingElements[diNrOfEMS_OUT,arrCTCheckActivePrio[3]].arrTargetPowerEMS[5] > 0 OR Lynus_Standards.GVL_Energy.stDataElectricHeatingElements[diNrOfEMS_OUT,arrCTCheckActivePrio[3]].arrTargetPowerEMS[6] > 0) THEN
								IF Lynus_Standards.GVL_Energy.stDataElectricHeatingElements[diNrOfEMS_OUT,arrCTCheckActivePrio[3]].arrTargetPowerEMS[2] <= 0 THEN arrActualStepInTurn[2] := 1; END_IF
								IF Lynus_Standards.GVL_Energy.stDataElectricHeatingElements[diNrOfEMS_OUT,arrCTCheckActivePrio[3]].arrTargetPowerEMS[2] > 0 THEN arrActualStepInTurn[2] := 2; END_IF
								IF Lynus_Standards.GVL_Energy.stDataElectricHeatingElements[diNrOfEMS_OUT,arrCTCheckActivePrio[3]].arrTargetPowerEMS[3] > 0 THEN arrActualStepInTurn[2] := 3; END_IF
								IF Lynus_Standards.GVL_Energy.stDataElectricHeatingElements[diNrOfEMS_OUT,arrCTCheckActivePrio[3]].arrTargetPowerEMS[4] > 0 THEN arrActualStepInTurn[2] := 4; END_IF
								IF Lynus_Standards.GVL_Energy.stDataElectricHeatingElements[diNrOfEMS_OUT,arrCTCheckActivePrio[3]].arrTargetPowerEMS[5] > 0 THEN arrActualStepInTurn[2] := 5; END_IF
								IF Lynus_Standards.GVL_Energy.stDataElectricHeatingElements[diNrOfEMS_OUT,arrCTCheckActivePrio[3]].arrTargetPowerEMS[6] > 0 THEN arrActualStepInTurn[2] := 6; END_IF
									arrMaxPrioReached[3] := FALSE;
										arrMinPrioReached[3] := FALSE;
											arrCTCheckActivePrio[3] := 0;
												uiState := 90;
				ELSIF NOT bSurplusAvailable AND Lynus_Standards.GVL_Energy.stDataElectricHeatingElements[diNrOfEMS_OUT,arrCTCheckActivePrio[3]].byPriority = arrActualPrioInTurn[3] AND Lynus_Standards.GVL_Energy.stDataElectricHeatingElements[diNrOfEMS_OUT,arrCTCheckActivePrio[3]].bIsStepSwitched AND 
					Lynus_Standards.GVL_Energy.stDataElectricHeatingElements[diNrOfEMS_OUT,arrCTCheckActivePrio[3]].bIsControllable AND Lynus_Standards.GVL_Energy.stDataElectricHeatingElements[diNrOfEMS_OUT,arrCTCheckActivePrio[3]].byNumberOfSteps = 7 AND 
						(Lynus_Standards.GVL_Energy.stDataElectricHeatingElements[diNrOfEMS_OUT,arrCTCheckActivePrio[3]].arrTargetPowerEMS[1] > 0 OR Lynus_Standards.GVL_Energy.stDataElectricHeatingElements[diNrOfEMS_OUT,arrCTCheckActivePrio[3]].arrTargetPowerEMS[2] > 0 OR Lynus_Standards.GVL_Energy.stDataElectricHeatingElements[diNrOfEMS_OUT,arrCTCheckActivePrio[3]].arrTargetPowerEMS[3] > 0 OR
							Lynus_Standards.GVL_Energy.stDataElectricHeatingElements[diNrOfEMS_OUT,arrCTCheckActivePrio[3]].arrTargetPowerEMS[4] > 0 OR Lynus_Standards.GVL_Energy.stDataElectricHeatingElements[diNrOfEMS_OUT,arrCTCheckActivePrio[3]].arrTargetPowerEMS[5] > 0 OR Lynus_Standards.GVL_Energy.stDataElectricHeatingElements[diNrOfEMS_OUT,arrCTCheckActivePrio[3]].arrTargetPowerEMS[6] > 0 OR
								Lynus_Standards.GVL_Energy.stDataElectricHeatingElements[diNrOfEMS_OUT,arrCTCheckActivePrio[3]].arrTargetPowerEMS[7] > 0) THEN
									IF Lynus_Standards.GVL_Energy.stDataElectricHeatingElements[diNrOfEMS_OUT,arrCTCheckActivePrio[3]].arrTargetPowerEMS[2] <= 0 THEN arrActualStepInTurn[2] := 1; END_IF
									IF Lynus_Standards.GVL_Energy.stDataElectricHeatingElements[diNrOfEMS_OUT,arrCTCheckActivePrio[3]].arrTargetPowerEMS[2] > 0 THEN arrActualStepInTurn[2] := 2; END_IF
									IF Lynus_Standards.GVL_Energy.stDataElectricHeatingElements[diNrOfEMS_OUT,arrCTCheckActivePrio[3]].arrTargetPowerEMS[3] > 0 THEN arrActualStepInTurn[2] := 3; END_IF
									IF Lynus_Standards.GVL_Energy.stDataElectricHeatingElements[diNrOfEMS_OUT,arrCTCheckActivePrio[3]].arrTargetPowerEMS[4] > 0 THEN arrActualStepInTurn[2] := 4; END_IF
									IF Lynus_Standards.GVL_Energy.stDataElectricHeatingElements[diNrOfEMS_OUT,arrCTCheckActivePrio[3]].arrTargetPowerEMS[5] > 0 THEN arrActualStepInTurn[2] := 5; END_IF
									IF Lynus_Standards.GVL_Energy.stDataElectricHeatingElements[diNrOfEMS_OUT,arrCTCheckActivePrio[3]].arrTargetPowerEMS[6] > 0 THEN arrActualStepInTurn[2] := 6; END_IF
									IF Lynus_Standards.GVL_Energy.stDataElectricHeatingElements[diNrOfEMS_OUT,arrCTCheckActivePrio[3]].arrTargetPowerEMS[7] > 0 THEN arrActualStepInTurn[2] := 7; END_IF
										arrMaxPrioReached[3] := FALSE;
											arrMinPrioReached[3] := FALSE;
												arrCTCheckActivePrio[3] := 0;
													uiState := 90;
				ELSIF NOT bSurplusAvailable AND Lynus_Standards.GVL_Energy.stDataElectricHeatingElements[diNrOfEMS_OUT,arrCTCheckActivePrio[3]].byPriority = arrActualPrioInTurn[3] AND Lynus_Standards.GVL_Energy.stDataElectricHeatingElements[diNrOfEMS_OUT,arrCTCheckActivePrio[3]].bIsStepSwitched AND 
					Lynus_Standards.GVL_Energy.stDataElectricHeatingElements[diNrOfEMS_OUT,arrCTCheckActivePrio[3]].bIsControllable AND Lynus_Standards.GVL_Energy.stDataElectricHeatingElements[diNrOfEMS_OUT,arrCTCheckActivePrio[3]].byNumberOfSteps = 8 AND 
						(Lynus_Standards.GVL_Energy.stDataElectricHeatingElements[diNrOfEMS_OUT,arrCTCheckActivePrio[3]].arrTargetPowerEMS[1] > 0 OR Lynus_Standards.GVL_Energy.stDataElectricHeatingElements[diNrOfEMS_OUT,arrCTCheckActivePrio[3]].arrTargetPowerEMS[2] > 0 OR Lynus_Standards.GVL_Energy.stDataElectricHeatingElements[diNrOfEMS_OUT,arrCTCheckActivePrio[3]].arrTargetPowerEMS[3] > 0 OR
							Lynus_Standards.GVL_Energy.stDataElectricHeatingElements[diNrOfEMS_OUT,arrCTCheckActivePrio[3]].arrTargetPowerEMS[4] > 0 OR Lynus_Standards.GVL_Energy.stDataElectricHeatingElements[diNrOfEMS_OUT,arrCTCheckActivePrio[3]].arrTargetPowerEMS[5] > 0 OR Lynus_Standards.GVL_Energy.stDataElectricHeatingElements[diNrOfEMS_OUT,arrCTCheckActivePrio[3]].arrTargetPowerEMS[6] > 0 OR
								Lynus_Standards.GVL_Energy.stDataElectricHeatingElements[diNrOfEMS_OUT,arrCTCheckActivePrio[3]].arrTargetPowerEMS[7] > 0 OR Lynus_Standards.GVL_Energy.stDataElectricHeatingElements[diNrOfEMS_OUT,arrCTCheckActivePrio[3]].arrTargetPowerEMS[8] > 0) THEN
									IF Lynus_Standards.GVL_Energy.stDataElectricHeatingElements[diNrOfEMS_OUT,arrCTCheckActivePrio[3]].arrTargetPowerEMS[2] <= 0 THEN arrActualStepInTurn[2] := 1; END_IF
									IF Lynus_Standards.GVL_Energy.stDataElectricHeatingElements[diNrOfEMS_OUT,arrCTCheckActivePrio[3]].arrTargetPowerEMS[2] > 0 THEN arrActualStepInTurn[2] := 2; END_IF
									IF Lynus_Standards.GVL_Energy.stDataElectricHeatingElements[diNrOfEMS_OUT,arrCTCheckActivePrio[3]].arrTargetPowerEMS[3] > 0 THEN arrActualStepInTurn[2] := 3; END_IF
									IF Lynus_Standards.GVL_Energy.stDataElectricHeatingElements[diNrOfEMS_OUT,arrCTCheckActivePrio[3]].arrTargetPowerEMS[4] > 0 THEN arrActualStepInTurn[2] := 4; END_IF
									IF Lynus_Standards.GVL_Energy.stDataElectricHeatingElements[diNrOfEMS_OUT,arrCTCheckActivePrio[3]].arrTargetPowerEMS[5] > 0 THEN arrActualStepInTurn[2] := 5; END_IF
									IF Lynus_Standards.GVL_Energy.stDataElectricHeatingElements[diNrOfEMS_OUT,arrCTCheckActivePrio[3]].arrTargetPowerEMS[6] > 0 THEN arrActualStepInTurn[2] := 6; END_IF
									IF Lynus_Standards.GVL_Energy.stDataElectricHeatingElements[diNrOfEMS_OUT,arrCTCheckActivePrio[3]].arrTargetPowerEMS[7] > 0 THEN arrActualStepInTurn[2] := 7; END_IF
									IF Lynus_Standards.GVL_Energy.stDataElectricHeatingElements[diNrOfEMS_OUT,arrCTCheckActivePrio[3]].arrTargetPowerEMS[8] > 0 THEN arrActualStepInTurn[2] := 8; END_IF
										arrMaxPrioReached[3] := FALSE;
											arrMinPrioReached[3] := FALSE;
												arrCTCheckActivePrio[3] := 0;
													uiState := 90;
				ELSIF NOT bSurplusAvailable AND Lynus_Standards.GVL_Energy.stDataElectricHeatingElements[diNrOfEMS_OUT,arrCTCheckActivePrio[3]].byPriority = arrActualPrioInTurn[3] AND Lynus_Standards.GVL_Energy.stDataElectricHeatingElements[diNrOfEMS_OUT,arrCTCheckActivePrio[3]].bIsStepSwitched AND 
					Lynus_Standards.GVL_Energy.stDataElectricHeatingElements[diNrOfEMS_OUT,arrCTCheckActivePrio[3]].bIsControllable AND Lynus_Standards.GVL_Energy.stDataElectricHeatingElements[diNrOfEMS_OUT,arrCTCheckActivePrio[3]].byNumberOfSteps = 9 AND 
						(Lynus_Standards.GVL_Energy.stDataElectricHeatingElements[diNrOfEMS_OUT,arrCTCheckActivePrio[3]].arrTargetPowerEMS[1] > 0 OR Lynus_Standards.GVL_Energy.stDataElectricHeatingElements[diNrOfEMS_OUT,arrCTCheckActivePrio[3]].arrTargetPowerEMS[2] > 0 OR Lynus_Standards.GVL_Energy.stDataElectricHeatingElements[diNrOfEMS_OUT,arrCTCheckActivePrio[3]].arrTargetPowerEMS[3] > 0 OR
							Lynus_Standards.GVL_Energy.stDataElectricHeatingElements[diNrOfEMS_OUT,arrCTCheckActivePrio[3]].arrTargetPowerEMS[4] > 0 OR Lynus_Standards.GVL_Energy.stDataElectricHeatingElements[diNrOfEMS_OUT,arrCTCheckActivePrio[3]].arrTargetPowerEMS[5] > 0 OR Lynus_Standards.GVL_Energy.stDataElectricHeatingElements[diNrOfEMS_OUT,arrCTCheckActivePrio[3]].arrTargetPowerEMS[6] > 0 OR
								Lynus_Standards.GVL_Energy.stDataElectricHeatingElements[diNrOfEMS_OUT,arrCTCheckActivePrio[3]].arrTargetPowerEMS[7] > 0 OR Lynus_Standards.GVL_Energy.stDataElectricHeatingElements[diNrOfEMS_OUT,arrCTCheckActivePrio[3]].arrTargetPowerEMS[8] > 0 OR Lynus_Standards.GVL_Energy.stDataElectricHeatingElements[diNrOfEMS_OUT,arrCTCheckActivePrio[3]].arrTargetPowerEMS[9] > 0) THEN
									IF Lynus_Standards.GVL_Energy.stDataElectricHeatingElements[diNrOfEMS_OUT,arrCTCheckActivePrio[3]].arrTargetPowerEMS[2] <= 0 THEN arrActualStepInTurn[2] := 1; END_IF
									IF Lynus_Standards.GVL_Energy.stDataElectricHeatingElements[diNrOfEMS_OUT,arrCTCheckActivePrio[3]].arrTargetPowerEMS[2] > 0 THEN arrActualStepInTurn[2] := 2; END_IF
									IF Lynus_Standards.GVL_Energy.stDataElectricHeatingElements[diNrOfEMS_OUT,arrCTCheckActivePrio[3]].arrTargetPowerEMS[3] > 0 THEN arrActualStepInTurn[2] := 3; END_IF
									IF Lynus_Standards.GVL_Energy.stDataElectricHeatingElements[diNrOfEMS_OUT,arrCTCheckActivePrio[3]].arrTargetPowerEMS[4] > 0 THEN arrActualStepInTurn[2] := 4; END_IF
									IF Lynus_Standards.GVL_Energy.stDataElectricHeatingElements[diNrOfEMS_OUT,arrCTCheckActivePrio[3]].arrTargetPowerEMS[5] > 0 THEN arrActualStepInTurn[2] := 5; END_IF
									IF Lynus_Standards.GVL_Energy.stDataElectricHeatingElements[diNrOfEMS_OUT,arrCTCheckActivePrio[3]].arrTargetPowerEMS[6] > 0 THEN arrActualStepInTurn[2] := 6; END_IF
									IF Lynus_Standards.GVL_Energy.stDataElectricHeatingElements[diNrOfEMS_OUT,arrCTCheckActivePrio[3]].arrTargetPowerEMS[7] > 0 THEN arrActualStepInTurn[2] := 7; END_IF
									IF Lynus_Standards.GVL_Energy.stDataElectricHeatingElements[diNrOfEMS_OUT,arrCTCheckActivePrio[3]].arrTargetPowerEMS[8] > 0 THEN arrActualStepInTurn[2] := 8; END_IF
									IF Lynus_Standards.GVL_Energy.stDataElectricHeatingElements[diNrOfEMS_OUT,arrCTCheckActivePrio[3]].arrTargetPowerEMS[9] > 0 THEN arrActualStepInTurn[2] := 9; END_IF
										arrMaxPrioReached[3] := FALSE;
											arrMinPrioReached[3] := FALSE;
												arrCTCheckActivePrio[3] := 0;
													uiState := 90;
				ELSIF NOT bSurplusAvailable AND Lynus_Standards.GVL_Energy.stDataElectricHeatingElements[diNrOfEMS_OUT,arrCTCheckActivePrio[3]].byPriority = arrActualPrioInTurn[3] AND Lynus_Standards.GVL_Energy.stDataElectricHeatingElements[diNrOfEMS_OUT,arrCTCheckActivePrio[3]].bIsStepSwitched AND 
					Lynus_Standards.GVL_Energy.stDataElectricHeatingElements[diNrOfEMS_OUT,arrCTCheckActivePrio[3]].bIsControllable AND Lynus_Standards.GVL_Energy.stDataElectricHeatingElements[diNrOfEMS_OUT,arrCTCheckActivePrio[3]].byNumberOfSteps = 10 AND 
						(Lynus_Standards.GVL_Energy.stDataElectricHeatingElements[diNrOfEMS_OUT,arrCTCheckActivePrio[3]].arrTargetPowerEMS[1] > 0 OR Lynus_Standards.GVL_Energy.stDataElectricHeatingElements[diNrOfEMS_OUT,arrCTCheckActivePrio[3]].arrTargetPowerEMS[2] > 0 OR Lynus_Standards.GVL_Energy.stDataElectricHeatingElements[diNrOfEMS_OUT,arrCTCheckActivePrio[3]].arrTargetPowerEMS[3] > 0 OR
							Lynus_Standards.GVL_Energy.stDataElectricHeatingElements[diNrOfEMS_OUT,arrCTCheckActivePrio[3]].arrTargetPowerEMS[4] > 0 OR Lynus_Standards.GVL_Energy.stDataElectricHeatingElements[diNrOfEMS_OUT,arrCTCheckActivePrio[3]].arrTargetPowerEMS[5] > 0 OR Lynus_Standards.GVL_Energy.stDataElectricHeatingElements[diNrOfEMS_OUT,arrCTCheckActivePrio[3]].arrTargetPowerEMS[6] > 0 OR
								Lynus_Standards.GVL_Energy.stDataElectricHeatingElements[diNrOfEMS_OUT,arrCTCheckActivePrio[3]].arrTargetPowerEMS[7] > 0 OR Lynus_Standards.GVL_Energy.stDataElectricHeatingElements[diNrOfEMS_OUT,arrCTCheckActivePrio[3]].arrTargetPowerEMS[8] > 0 OR Lynus_Standards.GVL_Energy.stDataElectricHeatingElements[diNrOfEMS_OUT,arrCTCheckActivePrio[3]].arrTargetPowerEMS[9] > 0 OR
									Lynus_Standards.GVL_Energy.stDataElectricHeatingElements[diNrOfEMS_OUT,arrCTCheckActivePrio[3]].arrTargetPowerEMS[10] > 0) THEN
										IF Lynus_Standards.GVL_Energy.stDataElectricHeatingElements[diNrOfEMS_OUT,arrCTCheckActivePrio[3]].arrTargetPowerEMS[2] <= 0 THEN arrActualStepInTurn[2] := 1; END_IF
										IF Lynus_Standards.GVL_Energy.stDataElectricHeatingElements[diNrOfEMS_OUT,arrCTCheckActivePrio[3]].arrTargetPowerEMS[2] > 0 THEN arrActualStepInTurn[2] := 2; END_IF
										IF Lynus_Standards.GVL_Energy.stDataElectricHeatingElements[diNrOfEMS_OUT,arrCTCheckActivePrio[3]].arrTargetPowerEMS[3] > 0 THEN arrActualStepInTurn[2] := 3; END_IF
										IF Lynus_Standards.GVL_Energy.stDataElectricHeatingElements[diNrOfEMS_OUT,arrCTCheckActivePrio[3]].arrTargetPowerEMS[4] > 0 THEN arrActualStepInTurn[2] := 4; END_IF
										IF Lynus_Standards.GVL_Energy.stDataElectricHeatingElements[diNrOfEMS_OUT,arrCTCheckActivePrio[3]].arrTargetPowerEMS[5] > 0 THEN arrActualStepInTurn[2] := 5; END_IF
										IF Lynus_Standards.GVL_Energy.stDataElectricHeatingElements[diNrOfEMS_OUT,arrCTCheckActivePrio[3]].arrTargetPowerEMS[6] > 0 THEN arrActualStepInTurn[2] := 6; END_IF
										IF Lynus_Standards.GVL_Energy.stDataElectricHeatingElements[diNrOfEMS_OUT,arrCTCheckActivePrio[3]].arrTargetPowerEMS[7] > 0 THEN arrActualStepInTurn[2] := 7; END_IF
										IF Lynus_Standards.GVL_Energy.stDataElectricHeatingElements[diNrOfEMS_OUT,arrCTCheckActivePrio[3]].arrTargetPowerEMS[8] > 0 THEN arrActualStepInTurn[2] := 8; END_IF
										IF Lynus_Standards.GVL_Energy.stDataElectricHeatingElements[diNrOfEMS_OUT,arrCTCheckActivePrio[3]].arrTargetPowerEMS[9] > 0 THEN arrActualStepInTurn[2] := 9; END_IF
										IF Lynus_Standards.GVL_Energy.stDataElectricHeatingElements[diNrOfEMS_OUT,arrCTCheckActivePrio[3]].arrTargetPowerEMS[10] > 0 THEN arrActualStepInTurn[2] := 10; END_IF
											arrMaxPrioReached[3] := FALSE;
												arrMinPrioReached[3] := FALSE;
													arrCTCheckActivePrio[3] := 0;
														uiState := 90;
				ELSE
					IF NOT bSurplusAvailable AND arrActualPrioInTurn[3] > 1 AND uiState = 70 AND arrCTCheckActivePrio[3] = Constants_Energy.diMaxNumberOfElectricHeatingElements THEN 
						arrActualPrioInTurn[3] := arrActualPrioInTurn[3] - 1; arrCTCheckActivePrio[3] := 0; liCounterCkeckDeviceAndPrio := 0; liNrOfNotDoneDevices := 0; 
					END_IF
				END_IF
		
		//Go to next step if we are on min prio or on max prio and the target power is just set to the min or to the max value.
		liCounterCkeckDeviceAndPrio := LIMIT(1,liCounterCkeckDeviceAndPrio,Constants_Energy.diMaxNumberOfElectricHeatingElements);
		
			IF arrActualPrioInTurn[3] = 1 AND Lynus_Standards.GVL_Energy.stDataElectricHeatingElements[diNrOfEMS_OUT,liCounterCkeckDeviceAndPrio].byPriority = 1 AND
				(Lynus_Standards.GVL_Energy.stDataElectricHeatingElements[diNrOfEMS_OUT,liCounterCkeckDeviceAndPrio].arrTargetPowerEMS[1] <> 0 OR Lynus_Standards.GVL_Energy.stDataElectricHeatingElements[diNrOfEMS_OUT,liCounterCkeckDeviceAndPrio].arrTargetPowerEMS[2] <> 0 OR
					Lynus_Standards.GVL_Energy.stDataElectricHeatingElements[diNrOfEMS_OUT,liCounterCkeckDeviceAndPrio].arrTargetPowerEMS[3] <> 0 OR Lynus_Standards.GVL_Energy.stDataElectricHeatingElements[diNrOfEMS_OUT,liCounterCkeckDeviceAndPrio].arrTargetPowerEMS[4] <> 0 OR
						Lynus_Standards.GVL_Energy.stDataElectricHeatingElements[diNrOfEMS_OUT,liCounterCkeckDeviceAndPrio].arrTargetPowerEMS[5] <> 0 OR Lynus_Standards.GVL_Energy.stDataElectricHeatingElements[diNrOfEMS_OUT,liCounterCkeckDeviceAndPrio].arrTargetPowerEMS[6] <> 0 OR
							Lynus_Standards.GVL_Energy.stDataElectricHeatingElements[diNrOfEMS_OUT,liCounterCkeckDeviceAndPrio].arrTargetPowerEMS[7] <> 0 OR Lynus_Standards.GVL_Energy.stDataElectricHeatingElements[diNrOfEMS_OUT,liCounterCkeckDeviceAndPrio].arrTargetPowerEMS[8] <> 0 OR
								Lynus_Standards.GVL_Energy.stDataElectricHeatingElements[diNrOfEMS_OUT,liCounterCkeckDeviceAndPrio].arrTargetPowerEMS[9] <> 0 OR Lynus_Standards.GVL_Energy.stDataElectricHeatingElements[diNrOfEMS_OUT,liCounterCkeckDeviceAndPrio].arrTargetPowerEMS[10] <> 0) THEN 
									liNrOfNotDoneDevices := liNrOfNotDoneDevices + 1; 
			END_IF
				//1 Step
				IF arrActualPrioInTurn[3] = 255 AND Lynus_Standards.GVL_Energy.stDataElectricHeatingElements[diNrOfEMS_OUT,liCounterCkeckDeviceAndPrio].byPriority = 255 AND Lynus_Standards.GVL_Energy.stDataElectricHeatingElements[diNrOfEMS_OUT,liCounterCkeckDeviceAndPrio].byNumberOfSteps = 1 AND 
					Lynus_Standards.GVL_Energy.stDataElectricHeatingElements[diNrOfEMS_OUT,liCounterCkeckDeviceAndPrio].arrTargetPowerEMS[1] < 100 THEN 
						liNrOfNotDoneDevices := liNrOfNotDoneDevices + 1; 
				//2 Steps
				ELSIF arrActualPrioInTurn[3] = 255 AND Lynus_Standards.GVL_Energy.stDataElectricHeatingElements[diNrOfEMS_OUT,liCounterCkeckDeviceAndPrio].byPriority = 255 AND Lynus_Standards.GVL_Energy.stDataElectricHeatingElements[diNrOfEMS_OUT,liCounterCkeckDeviceAndPrio].byNumberOfSteps = 2 AND 
					(Lynus_Standards.GVL_Energy.stDataElectricHeatingElements[diNrOfEMS_OUT,liCounterCkeckDeviceAndPrio].arrTargetPowerEMS[1] < 100 OR Lynus_Standards.GVL_Energy.stDataElectricHeatingElements[diNrOfEMS_OUT,liCounterCkeckDeviceAndPrio].arrTargetPowerEMS[2] < 100) THEN 
						liNrOfNotDoneDevices := liNrOfNotDoneDevices + 1; 
				//3 Steps
				ELSIF arrActualPrioInTurn[3] = 255 AND Lynus_Standards.GVL_Energy.stDataElectricHeatingElements[diNrOfEMS_OUT,liCounterCkeckDeviceAndPrio].byPriority = 255 AND Lynus_Standards.GVL_Energy.stDataElectricHeatingElements[diNrOfEMS_OUT,liCounterCkeckDeviceAndPrio].byNumberOfSteps = 3 AND 
					(Lynus_Standards.GVL_Energy.stDataElectricHeatingElements[diNrOfEMS_OUT,liCounterCkeckDeviceAndPrio].arrTargetPowerEMS[1] < 100 OR Lynus_Standards.GVL_Energy.stDataElectricHeatingElements[diNrOfEMS_OUT,liCounterCkeckDeviceAndPrio].arrTargetPowerEMS[2] < 100 OR
						Lynus_Standards.GVL_Energy.stDataElectricHeatingElements[diNrOfEMS_OUT,liCounterCkeckDeviceAndPrio].arrTargetPowerEMS[3] < 100) THEN 
							liNrOfNotDoneDevices := liNrOfNotDoneDevices + 1;
				//4 Steps
				ELSIF arrActualPrioInTurn[3] = 255 AND Lynus_Standards.GVL_Energy.stDataElectricHeatingElements[diNrOfEMS_OUT,liCounterCkeckDeviceAndPrio].byPriority = 255 AND Lynus_Standards.GVL_Energy.stDataElectricHeatingElements[diNrOfEMS_OUT,liCounterCkeckDeviceAndPrio].byNumberOfSteps = 4 AND 
					(Lynus_Standards.GVL_Energy.stDataElectricHeatingElements[diNrOfEMS_OUT,liCounterCkeckDeviceAndPrio].arrTargetPowerEMS[1] < 100 OR Lynus_Standards.GVL_Energy.stDataElectricHeatingElements[diNrOfEMS_OUT,liCounterCkeckDeviceAndPrio].arrTargetPowerEMS[2] < 100 OR
						Lynus_Standards.GVL_Energy.stDataElectricHeatingElements[diNrOfEMS_OUT,liCounterCkeckDeviceAndPrio].arrTargetPowerEMS[3] < 100 OR Lynus_Standards.GVL_Energy.stDataElectricHeatingElements[diNrOfEMS_OUT,liCounterCkeckDeviceAndPrio].arrTargetPowerEMS[4] < 100) THEN 
							liNrOfNotDoneDevices := liNrOfNotDoneDevices + 1;  
				//5 Steps
				ELSIF arrActualPrioInTurn[3] = 255 AND Lynus_Standards.GVL_Energy.stDataElectricHeatingElements[diNrOfEMS_OUT,liCounterCkeckDeviceAndPrio].byPriority = 255 AND Lynus_Standards.GVL_Energy.stDataElectricHeatingElements[diNrOfEMS_OUT,liCounterCkeckDeviceAndPrio].byNumberOfSteps = 5 AND 
					(Lynus_Standards.GVL_Energy.stDataElectricHeatingElements[diNrOfEMS_OUT,liCounterCkeckDeviceAndPrio].arrTargetPowerEMS[1] < 100 OR Lynus_Standards.GVL_Energy.stDataElectricHeatingElements[diNrOfEMS_OUT,liCounterCkeckDeviceAndPrio].arrTargetPowerEMS[2] < 100 OR
						Lynus_Standards.GVL_Energy.stDataElectricHeatingElements[diNrOfEMS_OUT,liCounterCkeckDeviceAndPrio].arrTargetPowerEMS[3] < 100 OR Lynus_Standards.GVL_Energy.stDataElectricHeatingElements[diNrOfEMS_OUT,liCounterCkeckDeviceAndPrio].arrTargetPowerEMS[4] < 100 OR
							Lynus_Standards.GVL_Energy.stDataElectricHeatingElements[diNrOfEMS_OUT,liCounterCkeckDeviceAndPrio].arrTargetPowerEMS[5] < 100) THEN 
								liNrOfNotDoneDevices := liNrOfNotDoneDevices + 1; 
				//6 Steps
				ELSIF arrActualPrioInTurn[3] = 255 AND Lynus_Standards.GVL_Energy.stDataElectricHeatingElements[diNrOfEMS_OUT,liCounterCkeckDeviceAndPrio].byPriority = 255 AND Lynus_Standards.GVL_Energy.stDataElectricHeatingElements[diNrOfEMS_OUT,liCounterCkeckDeviceAndPrio].byNumberOfSteps = 6 AND 
					(Lynus_Standards.GVL_Energy.stDataElectricHeatingElements[diNrOfEMS_OUT,liCounterCkeckDeviceAndPrio].arrTargetPowerEMS[1] < 100 OR Lynus_Standards.GVL_Energy.stDataElectricHeatingElements[diNrOfEMS_OUT,liCounterCkeckDeviceAndPrio].arrTargetPowerEMS[2] < 100 OR
						Lynus_Standards.GVL_Energy.stDataElectricHeatingElements[diNrOfEMS_OUT,liCounterCkeckDeviceAndPrio].arrTargetPowerEMS[3] < 100 OR Lynus_Standards.GVL_Energy.stDataElectricHeatingElements[diNrOfEMS_OUT,liCounterCkeckDeviceAndPrio].arrTargetPowerEMS[4] < 100 OR
							Lynus_Standards.GVL_Energy.stDataElectricHeatingElements[diNrOfEMS_OUT,liCounterCkeckDeviceAndPrio].arrTargetPowerEMS[5] < 100 OR Lynus_Standards.GVL_Energy.stDataElectricHeatingElements[diNrOfEMS_OUT,liCounterCkeckDeviceAndPrio].arrTargetPowerEMS[6] < 100) THEN 
								liNrOfNotDoneDevices := liNrOfNotDoneDevices + 1; 
				//7 Steps
				ELSIF arrActualPrioInTurn[3] = 255 AND Lynus_Standards.GVL_Energy.stDataElectricHeatingElements[diNrOfEMS_OUT,liCounterCkeckDeviceAndPrio].byPriority = 255 AND Lynus_Standards.GVL_Energy.stDataElectricHeatingElements[diNrOfEMS_OUT,liCounterCkeckDeviceAndPrio].byNumberOfSteps = 7 AND 
					(Lynus_Standards.GVL_Energy.stDataElectricHeatingElements[diNrOfEMS_OUT,liCounterCkeckDeviceAndPrio].arrTargetPowerEMS[1] < 100 OR Lynus_Standards.GVL_Energy.stDataElectricHeatingElements[diNrOfEMS_OUT,liCounterCkeckDeviceAndPrio].arrTargetPowerEMS[2] < 100 OR
						Lynus_Standards.GVL_Energy.stDataElectricHeatingElements[diNrOfEMS_OUT,liCounterCkeckDeviceAndPrio].arrTargetPowerEMS[3] < 100 OR Lynus_Standards.GVL_Energy.stDataElectricHeatingElements[diNrOfEMS_OUT,liCounterCkeckDeviceAndPrio].arrTargetPowerEMS[4] < 100 OR
							Lynus_Standards.GVL_Energy.stDataElectricHeatingElements[diNrOfEMS_OUT,liCounterCkeckDeviceAndPrio].arrTargetPowerEMS[5] < 100 OR Lynus_Standards.GVL_Energy.stDataElectricHeatingElements[diNrOfEMS_OUT,liCounterCkeckDeviceAndPrio].arrTargetPowerEMS[6] < 100 OR
								Lynus_Standards.GVL_Energy.stDataElectricHeatingElements[diNrOfEMS_OUT,liCounterCkeckDeviceAndPrio].arrTargetPowerEMS[7] < 100) THEN 
									liNrOfNotDoneDevices := liNrOfNotDoneDevices + 1; 
				//8 Steps
				ELSIF arrActualPrioInTurn[3] = 255 AND Lynus_Standards.GVL_Energy.stDataElectricHeatingElements[diNrOfEMS_OUT,liCounterCkeckDeviceAndPrio].byPriority = 255 AND Lynus_Standards.GVL_Energy.stDataElectricHeatingElements[diNrOfEMS_OUT,liCounterCkeckDeviceAndPrio].byNumberOfSteps = 8 AND 
					(Lynus_Standards.GVL_Energy.stDataElectricHeatingElements[diNrOfEMS_OUT,liCounterCkeckDeviceAndPrio].arrTargetPowerEMS[1] < 100 OR Lynus_Standards.GVL_Energy.stDataElectricHeatingElements[diNrOfEMS_OUT,liCounterCkeckDeviceAndPrio].arrTargetPowerEMS[2] < 100 OR
						Lynus_Standards.GVL_Energy.stDataElectricHeatingElements[diNrOfEMS_OUT,liCounterCkeckDeviceAndPrio].arrTargetPowerEMS[3] < 100 OR Lynus_Standards.GVL_Energy.stDataElectricHeatingElements[diNrOfEMS_OUT,liCounterCkeckDeviceAndPrio].arrTargetPowerEMS[4] < 100 OR
							Lynus_Standards.GVL_Energy.stDataElectricHeatingElements[diNrOfEMS_OUT,liCounterCkeckDeviceAndPrio].arrTargetPowerEMS[5] < 100 OR Lynus_Standards.GVL_Energy.stDataElectricHeatingElements[diNrOfEMS_OUT,liCounterCkeckDeviceAndPrio].arrTargetPowerEMS[6] < 100 OR
								Lynus_Standards.GVL_Energy.stDataElectricHeatingElements[diNrOfEMS_OUT,liCounterCkeckDeviceAndPrio].arrTargetPowerEMS[7] < 100 OR Lynus_Standards.GVL_Energy.stDataElectricHeatingElements[diNrOfEMS_OUT,liCounterCkeckDeviceAndPrio].arrTargetPowerEMS[8] < 100) THEN 
									liNrOfNotDoneDevices := liNrOfNotDoneDevices + 1; 
				//9 Steps
				ELSIF arrActualPrioInTurn[3] = 255 AND Lynus_Standards.GVL_Energy.stDataElectricHeatingElements[diNrOfEMS_OUT,liCounterCkeckDeviceAndPrio].byPriority = 255 AND Lynus_Standards.GVL_Energy.stDataElectricHeatingElements[diNrOfEMS_OUT,liCounterCkeckDeviceAndPrio].byNumberOfSteps = 9 AND 
					(Lynus_Standards.GVL_Energy.stDataElectricHeatingElements[diNrOfEMS_OUT,liCounterCkeckDeviceAndPrio].arrTargetPowerEMS[1] < 100 OR Lynus_Standards.GVL_Energy.stDataElectricHeatingElements[diNrOfEMS_OUT,liCounterCkeckDeviceAndPrio].arrTargetPowerEMS[2] < 100 OR
						Lynus_Standards.GVL_Energy.stDataElectricHeatingElements[diNrOfEMS_OUT,liCounterCkeckDeviceAndPrio].arrTargetPowerEMS[3] < 100 OR Lynus_Standards.GVL_Energy.stDataElectricHeatingElements[diNrOfEMS_OUT,liCounterCkeckDeviceAndPrio].arrTargetPowerEMS[4] < 100 OR
							Lynus_Standards.GVL_Energy.stDataElectricHeatingElements[diNrOfEMS_OUT,liCounterCkeckDeviceAndPrio].arrTargetPowerEMS[5] < 100 OR Lynus_Standards.GVL_Energy.stDataElectricHeatingElements[diNrOfEMS_OUT,liCounterCkeckDeviceAndPrio].arrTargetPowerEMS[6] < 100 OR
								Lynus_Standards.GVL_Energy.stDataElectricHeatingElements[diNrOfEMS_OUT,liCounterCkeckDeviceAndPrio].arrTargetPowerEMS[7] < 100 OR Lynus_Standards.GVL_Energy.stDataElectricHeatingElements[diNrOfEMS_OUT,liCounterCkeckDeviceAndPrio].arrTargetPowerEMS[8] < 100 OR
									Lynus_Standards.GVL_Energy.stDataElectricHeatingElements[diNrOfEMS_OUT,liCounterCkeckDeviceAndPrio].arrTargetPowerEMS[9] < 100) THEN 
										liNrOfNotDoneDevices := liNrOfNotDoneDevices + 1; 
				//10 Steps
				ELSIF arrActualPrioInTurn[3] = 255 AND Lynus_Standards.GVL_Energy.stDataElectricHeatingElements[diNrOfEMS_OUT,liCounterCkeckDeviceAndPrio].byPriority = 255 AND Lynus_Standards.GVL_Energy.stDataElectricHeatingElements[diNrOfEMS_OUT,liCounterCkeckDeviceAndPrio].byNumberOfSteps = 10 AND 
					(Lynus_Standards.GVL_Energy.stDataElectricHeatingElements[diNrOfEMS_OUT,liCounterCkeckDeviceAndPrio].arrTargetPowerEMS[1] < 100 OR Lynus_Standards.GVL_Energy.stDataElectricHeatingElements[diNrOfEMS_OUT,liCounterCkeckDeviceAndPrio].arrTargetPowerEMS[2] < 100 OR
						Lynus_Standards.GVL_Energy.stDataElectricHeatingElements[diNrOfEMS_OUT,liCounterCkeckDeviceAndPrio].arrTargetPowerEMS[3] < 100 OR Lynus_Standards.GVL_Energy.stDataElectricHeatingElements[diNrOfEMS_OUT,liCounterCkeckDeviceAndPrio].arrTargetPowerEMS[4] < 100 OR
							Lynus_Standards.GVL_Energy.stDataElectricHeatingElements[diNrOfEMS_OUT,liCounterCkeckDeviceAndPrio].arrTargetPowerEMS[5] < 100 OR Lynus_Standards.GVL_Energy.stDataElectricHeatingElements[diNrOfEMS_OUT,liCounterCkeckDeviceAndPrio].arrTargetPowerEMS[6] < 100 OR
								Lynus_Standards.GVL_Energy.stDataElectricHeatingElements[diNrOfEMS_OUT,liCounterCkeckDeviceAndPrio].arrTargetPowerEMS[7] < 100 OR Lynus_Standards.GVL_Energy.stDataElectricHeatingElements[diNrOfEMS_OUT,liCounterCkeckDeviceAndPrio].arrTargetPowerEMS[8] < 100 OR
									Lynus_Standards.GVL_Energy.stDataElectricHeatingElements[diNrOfEMS_OUT,liCounterCkeckDeviceAndPrio].arrTargetPowerEMS[9] < 100 OR Lynus_Standards.GVL_Energy.stDataElectricHeatingElements[diNrOfEMS_OUT,liCounterCkeckDeviceAndPrio].arrTargetPowerEMS[10] < 100) THEN 
										liNrOfNotDoneDevices := liNrOfNotDoneDevices + 1; 
				END_IF
		
		IF arrActualPrioInTurn[3] = 1 AND uiState = 70 AND liNrOfNotDoneDevices = 0 AND arrCTCheckActivePrio[3] = Constants_Energy.diMaxNumberOfElectricHeatingElements AND liCounterCkeckDeviceAndPrio = Constants_Energy.diMaxNumberOfElectricHeatingElements THEN 
			arrMinPrioReached[3] := TRUE; arrMaxPrioReached[3] := FALSE; liNrOfNotDoneDevices := 0; uiState := 90; arrCTCheckActivePrio[3] := 0; liCounterCkeckDeviceAndPrio := 0; 
		END_IF
		IF arrActualPrioInTurn[3] = 255 AND uiState = 70 AND liNrOfNotDoneDevices = 0 AND arrCTCheckActivePrio[3] = Constants_Energy.diMaxNumberOfElectricHeatingElements AND liCounterCkeckDeviceAndPrio = Constants_Energy.diMaxNumberOfElectricHeatingElements THEN 
			arrMaxPrioReached[3] := TRUE; arrMinPrioReached[3] := FALSE; liNrOfNotDoneDevices := 0; uiState := 90; arrCTCheckActivePrio[3] := 0; liCounterCkeckDeviceAndPrio := 0; 
		END_IF
		
		//Timout, go to next step
		IF timTimeout.Q AND uiState = 70 THEN uiState := 90; END_IF
		
	90: //Check the priority for the big consumer to controll it
		uiState_CP := uiState;
	
		//First check if we have min 1 of this Device Type. If not, complete this Device Type and go to the next step
		//Check also the bigest Priority of this Device Type
		diNumberOfDevicesFromEachType := 0; bySearchBigestPrio := 0;
		FOR liLPCheckDeviceAndPrio := 1 TO Constants_Energy.diMaxNumberOfOtherBigConsumers BY 1 DO
			IF Lynus_Standards.GVL_Energy.stDataOtherBigConsumers[diNrOfEMS_OUT,liLPCheckDeviceAndPrio].byPriority <> 0 THEN diNumberOfDevicesFromEachType := diNumberOfDevicesFromEachType + 1; END_IF
				IF Lynus_Standards.GVL_Energy.stDataOtherBigConsumers[diNrOfEMS_OUT,liLPCheckDeviceAndPrio].byPriority > bySearchBigestPrio THEN bySearchBigestPrio := Lynus_Standards.GVL_Energy.stDataOtherBigConsumers[diNrOfEMS_OUT,liLPCheckDeviceAndPrio].byPriority; END_IF   
		END_FOR 
			IF bSurplusAvailable AND arrActualPrioInTurn[4] > bySearchBigestPrio AND uiState = 90 THEN arrActualPrioInTurn[4] := 255; END_IF
				IF NOT bSurplusAvailable AND arrActualPrioInTurn[4] > bySearchBigestPrio AND uiState = 90 THEN arrActualPrioInTurn[4] := bySearchBigestPrio; END_IF
		
			IF bSurplusAvailable AND diNumberOfDevicesFromEachType = 0 THEN arrActualPrioInTurn[4] := 255; END_IF
				IF NOT bSurplusAvailable AND diNumberOfDevicesFromEachType = 0 THEN arrActualPrioInTurn[4] := 1; END_IF
		
		//Count up each Device
		arrCTCheckActivePrio[4] := arrCTCheckActivePrio[4] + 1;
			arrCTCheckActivePrio[4] := LIMIT(1,arrCTCheckActivePrio[4],Constants_Energy.diMaxNumberOfOtherBigConsumers);
		
			//Surplus
			IF bSurplusAvailable AND Lynus_Standards.GVL_Energy.stDataOtherBigConsumers[diNrOfEMS_OUT,arrCTCheckActivePrio[4]].byPriority = arrActualPrioInTurn[4] AND Lynus_Standards.GVL_Energy.stDataOtherBigConsumers[diNrOfEMS_OUT,arrCTCheckActivePrio[4]].rTargetPowerEMS < 100 THEN
				arrMaxPrioReached[4] := FALSE;
					arrMinPrioReached[4] := FALSE;
						arrCTCheckActivePrio[4] := 0;
							uiState := 109; 
			ELSE
				IF bSurplusAvailable AND arrActualPrioInTurn[4] < 255 AND uiState = 90 AND arrCTCheckActivePrio[4] = Constants_Energy.diMaxNumberOfOtherBigConsumers THEN arrActualPrioInTurn[4] := arrActualPrioInTurn[4] + 1; arrCTCheckActivePrio[4] := 0; END_IF
			END_IF
				//No surplus
				IF NOT bSurplusAvailable AND Lynus_Standards.GVL_Energy.stDataOtherBigConsumers[diNrOfEMS_OUT,arrCTCheckActivePrio[4]].byPriority = arrActualPrioInTurn[4] AND Lynus_Standards.GVL_Energy.stDataOtherBigConsumers[diNrOfEMS_OUT,arrCTCheckActivePrio[4]].rTargetPowerEMS > 0 THEN
					arrMaxPrioReached[4] := FALSE;
						arrMinPrioReached[4] := FALSE;
							arrCTCheckActivePrio[4] := 0;
								uiState := 109;
				ELSE
					IF NOT bSurplusAvailable AND arrActualPrioInTurn[4] > 1 AND uiState = 90 AND arrCTCheckActivePrio[4] = Constants_Energy.diMaxNumberOfOtherBigConsumers THEN arrActualPrioInTurn[4] := arrActualPrioInTurn[4] - 1; arrCTCheckActivePrio[4] := 0; END_IF
				END_IF
		
		
		//Go to next step if we are on min prio or on max prio and the target power is just set to the min or to the max value.
		liNrOfNotDoneDevices := 0;
			FOR liLPCheckDeviceAndPrio := 1 TO Constants_Energy.diMaxNumberOfOtherBigConsumers BY 1 DO
				IF arrActualPrioInTurn[4] = 1 AND Lynus_Standards.GVL_Energy.stDataOtherBigConsumers[diNrOfEMS_OUT,liLPCheckDeviceAndPrio].rTargetPowerEMS <> 0 AND Lynus_Standards.GVL_Energy.stDataOtherBigConsumers[diNrOfEMS_OUT,liLPCheckDeviceAndPrio].byPriority = 1 THEN
					liNrOfNotDoneDevices := liNrOfNotDoneDevices + 1;	
				END_IF
					IF arrActualPrioInTurn[4] = 255 AND Lynus_Standards.GVL_Energy.stDataOtherBigConsumers[diNrOfEMS_OUT,liLPCheckDeviceAndPrio].rTargetPowerEMS < 100 AND Lynus_Standards.GVL_Energy.stDataOtherBigConsumers[diNrOfEMS_OUT,liLPCheckDeviceAndPrio].byPriority = 255 THEN
						liNrOfNotDoneDevices := liNrOfNotDoneDevices + 1;	
					END_IF
			END_FOR	
		
		IF arrActualPrioInTurn[4] = 1 AND uiState = 90 AND liNrOfNotDoneDevices = 0 AND arrCTCheckActivePrio[4] = Constants_Energy.diMaxNumberOfOtherBigConsumers THEN 
			arrMinPrioReached[4] := TRUE; arrMaxPrioReached[4] := FALSE; liNrOfNotDoneDevices := 0; uiState := 109; arrCTCheckActivePrio[4] := 0; 
		END_IF
		IF arrActualPrioInTurn[4] = 255 AND uiState = 90 AND liNrOfNotDoneDevices = 0 AND arrCTCheckActivePrio[4] = Constants_Energy.diMaxNumberOfOtherBigConsumers THEN 
			arrMaxPrioReached[4] := TRUE; arrMinPrioReached[4] := FALSE; liNrOfNotDoneDevices := 0; uiState := 109; arrCTCheckActivePrio[4] := 0; 
		END_IF
		
		//Timout, go to next step
		IF timTimeout.Q AND uiState = 90 THEN uiState := 109; END_IF
		
	109://Check if in Load management mode or Peak shaving mode some electric Fuse Line use to much power when we have here surplus
		uiState_CP := uiState;

		//Count up each Device
		arrCTCheckActivePrio[5] := arrCTCheckActivePrio[5] + 1;
			arrCTCheckActivePrio[5] := LIMIT(1,arrCTCheckActivePrio[5],Constants_Energy.diMaxNumberOfElectricChargingStations);
		
		IF ((eOperationMode = E_OperatingMode_EMS.eLoadManagement OR eOperationMode = E_OperatingMode_EMS.ePeakLoadCapping) AND bSurplusAvailable AND stSetupEMS.bEnableMainFuseFunction) THEN
			IF Lynus_Standards.GVL_Energy.stDataElectricChargingStations[diNrOfEMS_OUT,arrCTCheckActivePrio[5]].byPriority = arrActualPrioInTurn[5] THEN
				//The ECS use to much power. So dont give here more power. Go to next priority
				IF bNoPowerForECS THEN
					//Go to next prio that we can go forward with the other Devices with same priority. Controlling for ECS see down on the Part on wich we limit the charging station about the electric Fuse Line
					IF arrActualPrioInTurn[5] < 255 THEN arrActualPrioInTurn[5] := arrActualPrioInTurn[5] + 1; END_IF
						uiState := 110;
							arrCTCheckActivePrio[5] := 0;	
				END_IF
			END_IF 
		ELSE
			uiState := 110;
				arrCTCheckActivePrio[5] := 0;
		END_IF
		
		//Go to next step if wa have checked every ECS without resluts
		IF arrCTCheckActivePrio[5] >= Constants_Energy.diMaxNumberOfElectricChargingStations AND uiState = 109 THEN
			uiState := 110;
				arrCTCheckActivePrio[5] := 0;
		END_IF 
	 	
		//Timout, go to next step
		IF timTimeout.Q AND uiState = 109 THEN uiState := 110; arrCTCheckActivePrio[5] := 0; END_IF	
		
	110: //Check the priority for the electric charging stations to controll it
		uiState_CP := uiState;
	
		//First check if we have min 1 of this Device Type. If not, complete this Device Type and go to the next step
		//Check also the bigest Priority of this Device Type
		diNumberOfDevicesFromEachType := 0; bySearchBigestPrio := 0;
		FOR liLPCheckDeviceAndPrio := 1 TO Constants_Energy.diMaxNumberOfElectricChargingStations BY 1 DO
			IF Lynus_Standards.GVL_Energy.stDataElectricChargingStations[diNrOfEMS_OUT,liLPCheckDeviceAndPrio].byPriority <> 0 THEN diNumberOfDevicesFromEachType := diNumberOfDevicesFromEachType + 1; END_IF
				IF Lynus_Standards.GVL_Energy.stDataElectricChargingStations[diNrOfEMS_OUT,liLPCheckDeviceAndPrio].byPriority > bySearchBigestPrio THEN bySearchBigestPrio := Lynus_Standards.GVL_Energy.stDataElectricChargingStations[diNrOfEMS_OUT,liLPCheckDeviceAndPrio].byPriority; END_IF   
		END_FOR 
			IF bSurplusAvailable AND arrActualPrioInTurn[5] > bySearchBigestPrio AND uiState = 110 THEN arrActualPrioInTurn[5] := 255; END_IF
				IF NOT bSurplusAvailable AND arrActualPrioInTurn[5] > bySearchBigestPrio AND uiState = 110 THEN arrActualPrioInTurn[5] := bySearchBigestPrio; END_IF
		
			IF bSurplusAvailable AND diNumberOfDevicesFromEachType = 0 THEN arrActualPrioInTurn[5] := 255; END_IF
				IF NOT bSurplusAvailable AND diNumberOfDevicesFromEachType = 0 THEN arrActualPrioInTurn[5] := 1; END_IF
		
		//Count up each Device
		arrCTCheckActivePrio[5] := arrCTCheckActivePrio[5] + 1;
			arrCTCheckActivePrio[5] := LIMIT(1,arrCTCheckActivePrio[5],Constants_Energy.diMaxNumberOfElectricChargingStations);
		
			//Surplus
			IF bSurplusAvailable AND Lynus_Standards.GVL_Energy.stDataElectricChargingStations[diNrOfEMS_OUT,arrCTCheckActivePrio[5]].byPriority = arrActualPrioInTurn[5] AND Lynus_Standards.GVL_Energy.stDataElectricChargingStations[diNrOfEMS_OUT,arrCTCheckActivePrio[5]].rTargetPowerEMS < 100 THEN
				arrMaxPrioReached[5] := FALSE;
					arrMinPrioReached[5] := FALSE;
						arrCTCheckActivePrio[5] := 0;
							uiState := 130;
			ELSE
				IF bSurplusAvailable AND arrActualPrioInTurn[5] < 255 AND uiState = 110 AND arrCTCheckActivePrio[5] = Constants_Energy.diMaxNumberOfElectricChargingStations THEN arrActualPrioInTurn[5] := arrActualPrioInTurn[5] + 1; arrCTCheckActivePrio[5] := 0; END_IF
			END_IF
				//No surplus
				IF NOT bSurplusAvailable AND Lynus_Standards.GVL_Energy.stDataElectricChargingStations[diNrOfEMS_OUT,arrCTCheckActivePrio[5]].byPriority = arrActualPrioInTurn[5] AND Lynus_Standards.GVL_Energy.stDataElectricChargingStations[diNrOfEMS_OUT,arrCTCheckActivePrio[5]].rTargetPowerEMS > 0 THEN
					arrMaxPrioReached[5] := FALSE;
						arrMinPrioReached[5] := FALSE;
							arrCTCheckActivePrio[5] := 0;
								uiState := 130;
				ELSE
					IF NOT bSurplusAvailable AND arrActualPrioInTurn[5] > 1 AND uiState = 110 AND arrCTCheckActivePrio[5] = Constants_Energy.diMaxNumberOfElectricChargingStations THEN arrActualPrioInTurn[5] := arrActualPrioInTurn[5] - 1; arrCTCheckActivePrio[5] := 0; END_IF
				END_IF
		
		//Go to next step if we are on min prio or on max prio and the target power is just set to the min or to the max value.
		liNrOfNotDoneDevices := 0;
			FOR liLPCheckDeviceAndPrio := 1 TO Constants_Energy.diMaxNumberOfElectricChargingStations BY 1 DO
				IF arrActualPrioInTurn[5] = 1 AND Lynus_Standards.GVL_Energy.stDataElectricChargingStations[diNrOfEMS_OUT,liLPCheckDeviceAndPrio].rTargetPowerEMS <> 0 AND Lynus_Standards.GVL_Energy.stDataElectricChargingStations[diNrOfEMS_OUT,liLPCheckDeviceAndPrio].byPriority = 1 THEN
					liNrOfNotDoneDevices := liNrOfNotDoneDevices + 1;	
				END_IF
					IF arrActualPrioInTurn[5] = 255 AND Lynus_Standards.GVL_Energy.stDataElectricChargingStations[diNrOfEMS_OUT,liLPCheckDeviceAndPrio].rTargetPowerEMS < 100 AND Lynus_Standards.GVL_Energy.stDataElectricChargingStations[diNrOfEMS_OUT,liLPCheckDeviceAndPrio].byPriority = 255 THEN
						liNrOfNotDoneDevices := liNrOfNotDoneDevices + 1;	
					END_IF
			END_FOR
		
		IF arrActualPrioInTurn[5] = 1 AND uiState = 110 AND liNrOfNotDoneDevices = 0 AND arrCTCheckActivePrio[5] = Constants_Energy.diMaxNumberOfElectricChargingStations THEN 
			arrMinPrioReached[5] := TRUE; arrMaxPrioReached[5] := FALSE; liNrOfNotDoneDevices := 0; uiState := 130; arrCTCheckActivePrio[5] := 0; 
		END_IF
		IF arrActualPrioInTurn[5] = 255 AND uiState = 110 AND liNrOfNotDoneDevices = 0 AND arrCTCheckActivePrio[5] = Constants_Energy.diMaxNumberOfElectricChargingStations THEN 
			arrMaxPrioReached[5] := TRUE; arrMinPrioReached[5] := FALSE; liNrOfNotDoneDevices := 0; uiState := 130; arrCTCheckActivePrio[5] := 0; 
		END_IF	
		
		//Timout, go to next step
		IF timTimeout.Q AND uiState = 110 THEN uiState := 130; END_IF
		
	130: //Search the smallest/biggest common priority and the number of devices with the same priority  
		IF bSurplusAvailable THEN bySmGrActiveCommonPrio := 255; END_IF
		IF NOT bSurplusAvailable THEN bySmGrActiveCommonPrio := 1; END_IF
	
		FOR byLPSmActiveCommonPrio := 1 TO 5 BY 1 DO
			IF bSurplusAvailable AND arrActualPrioInTurn[byLPSmActiveCommonPrio] < bySmGrActiveCommonPrio THEN bySmGrActiveCommonPrio := arrActualPrioInTurn[byLPSmActiveCommonPrio]; END_IF 
			IF NOT bSurplusAvailable AND arrActualPrioInTurn[byLPSmActiveCommonPrio] > bySmGrActiveCommonPrio THEN bySmGrActiveCommonPrio := arrActualPrioInTurn[byLPSmActiveCommonPrio]; END_IF 
		END_FOR
		
		//Back to the start when complete power is awarded, all power is set on 0 or we haven't common priority 	
		IF (arrMaxPrioReached[1] AND arrMaxPrioReached[2] AND arrMaxPrioReached[3] AND arrMaxPrioReached[4] AND arrMaxPrioReached[5]) OR
			(arrMinPrioReached[1] AND arrMinPrioReached[2] AND arrMinPrioReached[3] AND arrMinPrioReached[4] AND arrMinPrioReached[5]) THEN
				uiState := 10;
		ELSE
				uiState := 131;
		END_IF
		
	131: //Ckeck if the Batterys are full or not when we have no surplus. Thus the problem can be avoided if the battery FB regulates the power internally to 0, but the EMS still sends power to the inverter.
		 //Because otherwise it always takes too long when we have a small consumption and the battery must first be regulated to 0% in the GVL, although you are already full and you can therefore no longer be regulated back.
		 
		IF eOperationMode = E_OperatingMode_EMS.eSelfConsumption THEN 
			FOR liLPDataBatteryInverter := 1 TO Constants_Energy.diMaxNumberOfBatteryInverters BY 1 DO
				IF NOT bSurplusAvailable AND Lynus_Standards.GVL_Energy.stDataOfBatteryInverters[diNrOfEMS_OUT,liLPDataBatteryInverter].byPriority = bySmGrActiveCommonPrio AND 
					arrTimBatterysAreFull[liLPDataBatteryInverter].Q THEN
						Lynus_Standards.GVL_Energy.stDataOfBatteryInverters[diNrOfEMS_OUT,liLPDataBatteryInverter].rTargetPowerEMS := 0;
				END_IF	  
			END_FOR 
	
			//When we have a surplus again and the battery is full, we control it again with - 99.99%, so that the following devices do not have to wait too long to be controlled. 	
			//It must be set to 99.99, otherwise an error would occur in the next step.
			FOR liLPDataBatteryInverter := 1 TO Constants_Energy.diMaxNumberOfBatteryInverters BY 1 DO
				IF bSurplusAvailable AND Lynus_Standards.GVL_Energy.stDataOfBatteryInverters[diNrOfEMS_OUT,liLPDataBatteryInverter].byPriority = bySmGrActiveCommonPrio AND 
					arrTimBatterysAreFull[liLPDataBatteryInverter].Q THEN
						Lynus_Standards.GVL_Energy.stDataOfBatteryInverters[diNrOfEMS_OUT,liLPDataBatteryInverter].rTargetPowerEMS := - 99.99;
				END_IF	  
			END_FOR
		END_IF
		
		//Go to the next Step
		uiState := 150;
		
	150: //Calcualte the % power from each device with the same priority
		lrMaxPowerDevicesWithActualPrio := 0;
			bMissingPowerData := FALSE;
		
		//Batterys are only a "normal" Device, when the self consumption mode is active.
		IF eOperationMode = E_OperatingMode_EMS.eSelfConsumption THEN 
			//Batteryinverters
			FOR liLPCheckMaxPower := 1 TO Constants_Energy.diMaxNumberOfBatteryInverters BY 1 DO
				IF bSurplusAvailable AND Lynus_Standards.GVL_Energy.stDataOfBatteryInverters[diNrOfEMS_OUT,liLPCheckMaxPower].byPriority = bySmGrActiveCommonPrio AND Lynus_Standards.GVL_Energy.stDataOfBatteryInverters[diNrOfEMS_OUT,liLPCheckMaxPower].rTargetPowerEMS > -100 AND NOT Lynus_Standards.GVL_Energy.stDataOfBatteryInverters[diNrOfEMS_OUT,liLPCheckMaxPower].bWorkOnIslandMode THEN lrMaxPowerDevicesWithActualPrio := lrMaxPowerDevicesWithActualPrio + Lynus_Standards.GVL_Energy.stDataOfBatteryInverters[diNrOfEMS_OUT,liLPCheckMaxPower].rMaxChargePower; END_IF
				IF NOT bSurplusAvailable AND Lynus_Standards.GVL_Energy.stDataOfBatteryInverters[diNrOfEMS_OUT,liLPCheckMaxPower].byPriority = bySmGrActiveCommonPrio AND Lynus_Standards.GVL_Energy.stDataOfBatteryInverters[diNrOfEMS_OUT,liLPCheckMaxPower].rTargetPowerEMS < 0 AND NOT Lynus_Standards.GVL_Energy.stDataOfBatteryInverters[diNrOfEMS_OUT,liLPCheckMaxPower].bWorkOnIslandMode THEN lrMaxPowerDevicesWithActualPrio := lrMaxPowerDevicesWithActualPrio + Lynus_Standards.GVL_Energy.stDataOfBatteryInverters[diNrOfEMS_OUT,liLPCheckMaxPower].rMaxChargePower; END_IF 
			END_FOR
		END_IF
			//Heating pumps
			IF arrActualStepInTurn[1] >= 1 AND arrActualStepInTurn[1] <= 2 THEN
				FOR liLPCheckMaxPower := 1 TO Constants_Energy.diMaxNumberOfHeatingPumps BY 1 DO
					IF bSurplusAvailable AND Lynus_Standards.GVL_Energy.stDataHeatingPumps[diNrOfEMS_OUT,liLPCheckMaxPower].byPriority = bySmGrActiveCommonPrio AND Lynus_Standards.GVL_Energy.stDataHeatingPumps[diNrOfEMS_OUT,liLPCheckMaxPower].arrTargetPowerEMS[arrActualStepInTurn[1]] < 100 THEN lrMaxPowerDevicesWithActualPrio := lrMaxPowerDevicesWithActualPrio + Lynus_Standards.GVL_Energy.stDataHeatingPumps[diNrOfEMS_OUT,liLPCheckMaxPower].arrMaxPower[arrActualStepInTurn[1]]; END_IF
					IF NOT bSurplusAvailable AND Lynus_Standards.GVL_Energy.stDataHeatingPumps[diNrOfEMS_OUT,liLPCheckMaxPower].byPriority = bySmGrActiveCommonPrio AND Lynus_Standards.GVL_Energy.stDataHeatingPumps[diNrOfEMS_OUT,liLPCheckMaxPower].arrTargetPowerEMS[arrActualStepInTurn[1]] > 0 THEN lrMaxPowerDevicesWithActualPrio := lrMaxPowerDevicesWithActualPrio + Lynus_Standards.GVL_Energy.stDataHeatingPumps[diNrOfEMS_OUT,liLPCheckMaxPower].arrMaxPower[arrActualStepInTurn[1]]; END_IF
				END_FOR
			END_IF
				//Electric heating elements
				IF arrActualStepInTurn[2] >= 1 AND arrActualStepInTurn[2] <= 10 THEN
					FOR liLPCheckMaxPower := 1 TO Constants_Energy.diMaxNumberOfElectricHeatingElements BY 1 DO
						IF bSurplusAvailable AND Lynus_Standards.GVL_Energy.stDataElectricHeatingElements[diNrOfEMS_OUT,liLPCheckMaxPower].byPriority = bySmGrActiveCommonPrio AND Lynus_Standards.GVL_Energy.stDataElectricHeatingElements[diNrOfEMS_OUT,liLPCheckMaxPower].arrTargetPowerEMS[arrActualStepInTurn[2]] < 100 THEN lrMaxPowerDevicesWithActualPrio := lrMaxPowerDevicesWithActualPrio + Lynus_Standards.GVL_Energy.stDataElectricHeatingElements[diNrOfEMS_OUT,liLPCheckMaxPower].arrMaxPower[arrActualStepInTurn[2]]; END_IF 
						IF NOT bSurplusAvailable AND Lynus_Standards.GVL_Energy.stDataElectricHeatingElements[diNrOfEMS_OUT,liLPCheckMaxPower].byPriority = bySmGrActiveCommonPrio AND Lynus_Standards.GVL_Energy.stDataElectricHeatingElements[diNrOfEMS_OUT,liLPCheckMaxPower].arrTargetPowerEMS[arrActualStepInTurn[2]] > 0 THEN lrMaxPowerDevicesWithActualPrio := lrMaxPowerDevicesWithActualPrio + Lynus_Standards.GVL_Energy.stDataElectricHeatingElements[diNrOfEMS_OUT,liLPCheckMaxPower].arrMaxPower[arrActualStepInTurn[2]]; END_IF 
					END_FOR	
				END_IF
					//Other big consumer
					FOR liLPCheckMaxPower := 1 TO Constants_Energy.diMaxNumberOfOtherBigConsumers BY 1 DO
						IF bSurplusAvailable AND Lynus_Standards.GVL_Energy.stDataOtherBigConsumers[diNrOfEMS_OUT,liLPCheckMaxPower].byPriority = bySmGrActiveCommonPrio AND Lynus_Standards.GVL_Energy.stDataOtherBigConsumers[diNrOfEMS_OUT,liLPCheckMaxPower].rTargetPowerEMS < 100 THEN lrMaxPowerDevicesWithActualPrio := lrMaxPowerDevicesWithActualPrio + Lynus_Standards.GVL_Energy.stDataOtherBigConsumers[diNrOfEMS_OUT,liLPCheckMaxPower].rMaxPower; END_IF
						IF NOT bSurplusAvailable AND Lynus_Standards.GVL_Energy.stDataOtherBigConsumers[diNrOfEMS_OUT,liLPCheckMaxPower].byPriority = bySmGrActiveCommonPrio AND Lynus_Standards.GVL_Energy.stDataOtherBigConsumers[diNrOfEMS_OUT,liLPCheckMaxPower].rTargetPowerEMS > 0 THEN lrMaxPowerDevicesWithActualPrio := lrMaxPowerDevicesWithActualPrio + Lynus_Standards.GVL_Energy.stDataOtherBigConsumers[diNrOfEMS_OUT,liLPCheckMaxPower].rMaxPower; END_IF
					END_FOR
						//Electric charging stations
						FOR liLPCheckMaxPower := 1 TO Constants_Energy.diMaxNumberOfElectricChargingStations BY 1 DO
							IF bSurplusAvailable AND Lynus_Standards.GVL_Energy.stDataElectricChargingStations[diNrOfEMS_OUT,liLPCheckMaxPower].byPriority = bySmGrActiveCommonPrio AND Lynus_Standards.GVL_Energy.stDataElectricChargingStations[diNrOfEMS_OUT,liLPCheckMaxPower].rTargetPowerEMS < 100 THEN lrMaxPowerDevicesWithActualPrio := lrMaxPowerDevicesWithActualPrio + Lynus_Standards.GVL_Energy.stDataElectricChargingStations[diNrOfEMS_OUT,liLPCheckMaxPower].rMaxPower; END_IF
							IF NOT bSurplusAvailable AND Lynus_Standards.GVL_Energy.stDataElectricChargingStations[diNrOfEMS_OUT,liLPCheckMaxPower].byPriority = bySmGrActiveCommonPrio AND Lynus_Standards.GVL_Energy.stDataElectricChargingStations[diNrOfEMS_OUT,liLPCheckMaxPower].rTargetPowerEMS > 0 THEN lrMaxPowerDevicesWithActualPrio := lrMaxPowerDevicesWithActualPrio + Lynus_Standards.GVL_Energy.stDataElectricChargingStations[diNrOfEMS_OUT,liLPCheckMaxPower].rMaxPower; END_IF 
						END_FOR
		
		//Check is somthing has changed at the actual priority or at the actual step 
		//Priority or step now is higher as before
		IF (bSurplusAvailable AND MEMCMP(ADR(bySmGrActiveCommonPrio),ADR(bySmGrActiveCommonPrio_CP),SIZEOF(bySmGrActiveCommonPrio_CP)) <> 0) OR (bSurplusAvailable AND MEMCMP(ADR(arrActualStepInTurn),ADR(arrActualStepInTurn_CP),SIZEOF(arrActualStepInTurn_CP)) <> 0) THEN
			bySmGrActiveCommonPrio_CP := bySmGrActiveCommonPrio;
				arrActualStepInTurn_CP := arrActualStepInTurn;
					bStepWasOn100 := FALSE;		
		END_IF
			//Priority or step now is lower as before
			IF (NOT bSurplusAvailable AND MEMCMP(ADR(bySmGrActiveCommonPrio),ADR(bySmGrActiveCommonPrio_CP),SIZEOF(bySmGrActiveCommonPrio_CP)) <> 0) OR (NOT bSurplusAvailable AND MEMCMP(ADR(arrActualStepInTurn),ADR(arrActualStepInTurn_CP),SIZEOF(arrActualStepInTurn_CP)) <> 0) THEN
				bySmGrActiveCommonPrio_CP := bySmGrActiveCommonPrio;
					arrActualStepInTurn_CP := arrActualStepInTurn;
						bStepWasOn100 := TRUE;			
			END_IF						
						
		IF lrMaxPowerDevicesWithActualPrio > 0 THEN
			//Calcualte the power for the controllable devices
			IF bSurplusAvailable THEN rValuePercentToControllableDevices := LREAL_TO_REAL((100 * (lrActualSurplusOrConsumption * - 1)) / lrMaxPowerDevicesWithActualPrio); END_IF
  			IF NOT bSurplusAvailable THEN rValuePercentToControllableDevices := LREAL_TO_REAL((100 * lrActualSurplusOrConsumption) / lrMaxPowerDevicesWithActualPrio); END_IF
			//Calcualte the power for the On/Off or step switched devices
			IF bSurplusAvailable THEN rValuePercentToStepSwitchedDevices := LREAL_TO_REAL((100 * (lrActualSurplusOrConsumption * - 1)) / lrMaxPowerDevicesWithActualPrio); END_IF
			IF NOT bSurplusAvailable THEN rValuePercentToStepSwitchedDevices := (100 - LREAL_TO_REAL((100 * lrActualSurplusOrConsumption) / lrMaxPowerDevicesWithActualPrio)); END_IF
				IF bSurplusAvailable AND rValuePercentToStepSwitchedDevices >= 100 THEN bStepWasOn100 := TRUE; END_IF
				IF NOT bSurplusAvailable AND rValuePercentToStepSwitchedDevices < Constants_Energy.byTargetOffPowerForOnOffDevices THEN bStepWasOn100 := FALSE; END_IF
					IF bStepWasOn100 THEN rValuePercentToStepSwitchedDevices := 100; END_IF
					IF NOT bStepWasOn100 THEN rValuePercentToStepSwitchedDevices := 0; END_IF		
		ELSE
			//Power inputs from the setups of the devices are missing. Set the target power automatically to 0
			bMissingPowerData := TRUE;
			IF bSurplusAvailable THEN
				rValuePercentToControllableDevices := - 100;
				rValuePercentToStepSwitchedDevices := 0;
			END_IF
				IF NOT bSurplusAvailable THEN
					rValuePercentToControllableDevices := 100;
					rValuePercentToStepSwitchedDevices := 0;
				END_IF
		END_IF
		
		//If we have more surplus than the maximum power of the devices is, then we can set the target power directly to 100%
		IF bSurplusAvailable AND (lrActualSurplusOrConsumption * - 1) >= lrMaxPowerDevicesWithActualPrio AND NOT bMissingPowerData THEN rValuePercentToControllableDevices := 100; END_IF
		IF bSurplusAvailable AND (lrActualSurplusOrConsumption * - 1) >= lrMaxPowerDevicesWithActualPrio AND NOT bMissingPowerData THEN rValuePercentToStepSwitchedDevices := 100; bStepWasOn100 := TRUE; END_IF
		
		//If more power is consumed than the maximum power of the devices, 0% power can be commanded (for controllable devices 100% as it is deducted).
		IF NOT bSurplusAvailable AND lrActualSurplusOrConsumption >= lrMaxPowerDevicesWithActualPrio AND NOT bMissingPowerData THEN rValuePercentToControllableDevices := 100; END_IF
		IF NOT bSurplusAvailable AND lrActualSurplusOrConsumption >= lrMaxPowerDevicesWithActualPrio AND NOT bMissingPowerData THEN rValuePercentToStepSwitchedDevices := 0; bStepWasOn100 := FALSE; END_IF
		
		//Check the limits
		rValuePercentToControllableDevices := LIMIT(0,rValuePercentToControllableDevices,100);
			rValuePercentToStepSwitchedDevices := LIMIT(0,rValuePercentToStepSwitchedDevices,100);
				
		uiState := 170;
		
	170: //Set the target power to each device
		//Batterys or battery inverters
		//Batterys are only a "normal" Device, when the self consumption mode is active.
		IF eOperationMode = E_OperatingMode_EMS.eSelfConsumption THEN 
			FOR liLPSetPercentPower := 1 TO Constants_Energy.diMaxNumberOfBatteryInverters BY 1 DO
				IF bSurplusAvailable AND Lynus_Standards.GVL_Energy.stDataOfBatteryInverters[diNrOfEMS_OUT,liLPSetPercentPower].byPriority = bySmGrActiveCommonPrio AND Lynus_Standards.GVL_Energy.stDataOfBatteryInverters[diNrOfEMS_OUT,liLPSetPercentPower].rTargetPowerEMS > -100 THEN 
					Lynus_Standards.GVL_Energy.stDataOfBatteryInverters[diNrOfEMS_OUT,liLPSetPercentPower].rTargetPowerEMS := Lynus_Standards.GVL_Energy.stDataOfBatteryInverters[diNrOfEMS_OUT,liLPSetPercentPower].rTargetPowerEMS - rValuePercentToControllableDevices; 
				END_IF
				IF bSurplusAvailable AND Lynus_Standards.GVL_Energy.stDataOfBatteryInverters[diNrOfEMS_OUT,liLPSetPercentPower].rTargetPowerEMS < -100 THEN 
					Lynus_Standards.GVL_Energy.stDataOfBatteryInverters[diNrOfEMS_OUT,liLPSetPercentPower].rTargetPowerEMS := -100; 
				END_IF 
				IF NOT bSurplusAvailable AND Lynus_Standards.GVL_Energy.stDataOfBatteryInverters[diNrOfEMS_OUT,liLPSetPercentPower].byPriority = bySmGrActiveCommonPrio AND Lynus_Standards.GVL_Energy.stDataOfBatteryInverters[diNrOfEMS_OUT,liLPSetPercentPower].rTargetPowerEMS < 0 THEN 
					Lynus_Standards.GVL_Energy.stDataOfBatteryInverters[diNrOfEMS_OUT,liLPSetPercentPower].rTargetPowerEMS := Lynus_Standards.GVL_Energy.stDataOfBatteryInverters[diNrOfEMS_OUT,liLPSetPercentPower].rTargetPowerEMS + rValuePercentToControllableDevices;
				
				END_IF
				IF NOT bSurplusAvailable AND Lynus_Standards.GVL_Energy.stDataOfBatteryInverters[diNrOfEMS_OUT,liLPSetPercentPower].rTargetPowerEMS > 0 THEN 
					Lynus_Standards.GVL_Energy.stDataOfBatteryInverters[diNrOfEMS_OUT,liLPSetPercentPower].rTargetPowerEMS := 0;
					
